(* PLC project MQTT, CODESYS CODESYS V3.5 SP14, author Stefan Dreyer *)
(* stored: creationDateTime 2019-02-05T05:32:10.3765761, version 1.0.0.0, modificationDateTime 2019-02-04T05:34:23.4609065, organization Stefan Dreyer *)
(* MQTT Stuff
Using some cool stuff of OSCAT libs.
see oscat.de

more to describe *)

{attribute 'qualified_only'}
{attribute 'strict'}
TYPE INSERT_SPLIT_RETURN : (INSERT_NOT_VALID := 0, INSERT_DONE, INSERT_PENDING, INSERT_ERROR);
END_TYPE

TYPE MESSAGETYPE : (CONNECT := 16#10, CONNACK := 16#20, PUBLISH := 16#30, PUBACK := 16#40, PUBREC := 16#50, PUBREL := 16#60, PUBCOMP := 16#70, SUBSCRIBE := 16#80, SUBACK := 16#90, UNSUBSCRIBE := 16#A0, UNSUBACK := 16#B0, PINGREQ := 16#C0, PINGRESP := 16#D0, DISCONNECT := 16#E0) BYTE;
END_TYPE

{attribute 'qualified_only'}
{attribute 'strict'}
TYPE PROG_NUM : (Publish, Subscribe, ParseIncomming, MoveBuffer, ParsePublish, GetBufferFreePos, GetSplitTopic, DESTROY_HANDLE_MQTT, DESTROY_SPLIT_TOPIC, STATE_MASHINE_IN, STATE_MASHINE_OUT, SendOutData, SendInData, SendOutDataInsertTopic, SendOutDataInsertPayload);
END_TYPE

{attribute 'qualified_only'}
{attribute 'strict'}
TYPE PUSHOVER_SOUND : (Standart := 1);
END_TYPE

TYPE QoS : (AtMostOnce := 2#0, AtLeastOnce := 2#1, ExactlyOnce := 2#10, Fail := 2#10000000) BYTE;
END_TYPE

{attribute 'qualified_only'}
{attribute 'strict'}
TYPE STEPS_IN : (WAIT_DATA := 0, SEND_PUBACK, SEND_PUBREC, WAIT_PUBREL, SEND_PUBCOMP);
END_TYPE

{attribute 'qualified_only'}
{attribute 'strict'}
TYPE STEPS_OUT : (WAIT_DATA := 0, SEND_PUBLSIH, WAIT_PUBREC, SEND_PUBREL, WAIT_PUBCOMP, WAIT_PUBACK, WAIT_PINGRESP, SEND_SUBSCRIBE, WAIT_SUBACK, SEND_UNSUBSCRIBE, WAIT_UNSUBACK);
END_TYPE

{attribute 'qualified_only'}
{attribute 'strict'}
TYPE TOPIC_MATCH : (TOPIC_MATCHES := 1, TOPIC_DONT_MATCHES := 2) BYTE;
END_TYPE

{attribute 'qualified_only'}
{attribute 'strict'}
TYPE TOPIC_VALID : (TOPIC_UNTESTED := 0, TOPIC_VALID := 2, TOPIC_NOT_VALID := 1, TOPIC_NO_TEST := 3) BYTE;
END_TYPE

(* this data is passed to a subscription callback *)
TYPE CALLBACK_DATA : STRUCT
  PayloadString : POINTER TO STRING;  (* the Payload String *)
  Payload : POINTER TO BYTE;  (* pointer to binary payload *)
  PayloadSize : UDINT;  (* size of binary payload *)
  TopicOut : POINTER TO STRING;  (* here you get the compleete recived topic string *)
  TopicOutSplit : POINTER TO SPLIT_TOPIC;  (* split topic.... *)
  PayloadIsString : BOOL;  (* Payload is string *)
END_STRUCT;
END_TYPE

{attribute 'enable_dynamic_creation'}
TYPE CALLBACK_INSTANCES : STRUCT
  callback : MQTT_SUBSCRIBE_CALLBACK;
  next : POINTER TO CALLBACK_INSTANCES;
  last : BOOL := TRUE;
END_STRUCT;
END_TYPE

TYPE LIST_ALLVALUES_CALLBACK_DATA : STRUCT
  VarTYPE : CommonTypesAndFunctions.VAR_TYPES;
  Target : CommonTypesAndFunctions.ALL_TYPES_UNION_POINTER;
  SubTopic : POINTER TO STRING;  (* pointer to last subtopic or Payload Data to compare with *)
END_STRUCT;
END_TYPE

TYPE LIST_STRING_CALLBACK_DATA : STRUCT
  Target : POINTER TO STRING;  (* pointer to target string *)
  SubTopic : POINTER TO STRING;  (* pointer to last subtopic or Payload Data to compare with *)
END_STRUCT;
END_TYPE

TYPE MQTT_SUBSCRIBE_CALLBACKS : STRUCT
  Callback : MQTT_SUBSCRIBE_CALLBACK;
  FbId : UINT;
  ExpectingString : BOOL;  (* expecting string *)
  SplitTopic : POINTER TO HandleSplitTopic;
  free : BOOL := TRUE;  (* set to false if slot is aquired by an subscription *)
END_STRUCT;
END_TYPE

(* here the maximum sizes of paylod and topics are defined if dynamic low init of split topic is used, don't care about MaxTopicElementSize *)
TYPE COM_CONFIG : STRUCT
  MaxPayloadSize : UDINT := 2000;  (* max payload size *)
  MaxTopicLevels : UINT := 25;  (* max topic levels *)
  MaxTopicElementSize : UINT := 255;  (* Max Topic elemt size *)
END_STRUCT;
END_TYPE

TYPE DATA_FROM_BROKER : STRUCT
  MqttTopic : POINTER TO STRING;  (* use array in size of network buffer to split message dynamic, maybe not ... best is dynamic mammory.... or use an array of Pointer.... or callbacks so lets try to buffer public messages and releas one per cycle to application... now we try dynamic memmory.... MQTT Topic from Broker *)
  Topics : POINTER TO SPLIT_TOPIC;
  MqttPayload : POINTER TO BYTE;  (* MQTT Payload for Broker Payload from broker --> Pointer *)
  MqttPayloadSize : UDINT;  (* Payload size *)
  MessageType : MESSAGETYPE;  (* MQTT Message Type *)
  DataRecived : BOOL;  (* Data recived *)
END_STRUCT;
END_TYPE

TYPE DATA_TO_BROKER : STRUCT
  PaketData : PAKET_DATA;  (* Data of Paket *)
END_STRUCT;
END_TYPE

(* contro struct between HANDLE_MQTT and MQTT_CONTROL *)
TYPE MQTT_COM : STRUCT
  S_BUF : NETWORK_BUFFER;
  R_BUF : NETWORK_BUFFER;
  MQTT_CON : BOOL;  (* if falling edge close with disconnect packet *)
  MQTT_ABORT : BOOL;  (* if using this to disconnect, don't send disconnect paket.... *)
  MQTT_URL : STRING(OSCAT_BASIC.STRING_LENGTH);
  MQTT_PACKET_NO : WORD;
  TIMEOUT : TIME;
  TLS : BOOL;  (* DNS_IP4 : DWORD; set to true if you want to use TLS *)
  TLS_CONFIG : POINTER TO CommonTypesAndFunctions.TLS_CONFIG := 0;  (* data to TLS stuff *)
  MQTT_RCV_STATE : BYTE;  (* 0= non 1= recived 2= error *)
  ERROR_C : DWORD;
  ERROR_T : BYTE;
  CLIENT_ID : STRING(23);  (* CONNECT_TO_LOCALHOST:BOOL; *)
  CLIENT_WILL_TOPIC : STRING(255);  (* Topic vof will message after client id *)
  CLIENT_WILL_MESSAGE_DEAD : STRING(255);
  CLIENT_WILL_RETAIN : BOOL := TRUE;
  BROKER_USER : STRING(254);
  BROKER_PASSWORD : STRING(254);
  MQTT_NO_AWNSER : BOOL;  (* pakte wihout request-- return to recivestate 1 *)
END_STRUCT;
END_TYPE

TYPE MQTT_IN_DATA : STRUCT
  step : STEPS_IN;
  PaketID : WORD;
  WaitsForBuffFree : ULINT;
  TimeOut : ton;
  TimeOutStarted : BOOL;
  PUBLISHOrder : UINT;
  PUBCOMPOrder : UINT;
  QoS : QoS;
  CountPubrecRepeat : UINT;
END_STRUCT;
END_TYPE

TYPE MQTT_IN_OUT : STRUCT
  handleFB : POINTER TO HANDLE_MQTT;  (* pointer to handle FB *)
  In : POINTER TO PAKET_DATA;
  InFree : BOOL := TRUE;  (* in free, true if free *)
  TDI : CommonTypesAndFunctions.TIME_DATE_IMPULS_DATA;  (* time, date, impulse... *)
  TLS_CONFIG : POINTER TO CommonTypesAndFunctions.TLS_CONFIG := 0;  (* TLS stuff data *)
  BROKER_CONNECTED : BOOL;
  FB_NO_AUTO : UINT;
  FB_NO_AUTO_COUNT : UINT;  (* FBs count *)
  FB_NO_AUTO_TOKEN : UINT := 1;  (* FB Token *)
  COM_CONFIG : COM_CONFIG;  (* config for boot up *)
  ClientID : STRING(23) := 'CODESYS_MQTT';  (* client ID, only chars 0123456789abcdefghijklmnopqrstuvwxyzABCDEFGHIJKLMNOPQRSTUVWXYZ" System never can be anonymos *)
  WillTopicBase : STRING(255) := 'MQTTWill';
  ClientWillTopic : STRING(30) := 'DEAD';
  ClientWillMessage : STRING(30) := 'DIED';
  dynMemUsage : UDINT;  (* usage of dynamic RAM *)
  disconnectOnBufferOverflow : BOOL;  (* set this to one if you want the client to act like the standardt says if set to one and we receve mor publish pakets than we can handle, QoS 0 packets are lost and QoS 1 and 2 packets have to be repeaded by he broker *)
END_STRUCT;
END_TYPE

TYPE MQTT_INFO : STRUCT
  MQTT_CONNECTED : BOOL;
  MQTT_ERROR : STRING(OSCAT_BASIC.STRING_LENGTH);
END_STRUCT;
END_TYPE

TYPE MQTT_OUT_DATA : STRUCT
  InDataFromFb : POINTER TO PAKET_DATA;
  step : STEPS_OUT;
  WaitsForBuffFree : ULINT;
  PUBRECOrder : UINT;
  TimeOut : ton;
  TimeOutStarted : BOOL;
  PUBLISHOrder : UINT;
  PUBRELRepeatCounter : UINT;
END_STRUCT;
END_TYPE

TYPE PAKET_DATA : STRUCT
  MqttTopic : POINTER TO STRING;  (* MQTT Topic for Broker *)
  MqttTopicLength : UINT;  (* Topic length *)
  MqttPayload : POINTER TO BYTE;  (* MQTT Payload for Broker *)
  MqttPayloadLength : UDINT;  (* Payload length *)
  MessageType : MESSAGETYPE;  (* MQTT Message Type *)
  MessageQoS : QoS;  (* MQTT QoS *)
  SubackQoS : QoS;  (* SUCACK QoS Response *)
  MessageRetain : BOOL;  (* MQTT reatin *)
  DUP : BOOL;  (* Retry of paket *)
  PaketId : WORD;  (* PakatID for header *)
  FbId : UINT;  (* ID of MQTT FB to store or of request to Broker *)
  SendSucsess : BOOL;  (* Send was succsessfull *)
  Callback : MQTT_SUBSCRIBE_CALLBACK;  (* Callback FB for subscription *)
  SplitTopic : POINTER TO HandleSplitTopic;  (* split topic for subscribe *)
  CallbackError : BOOL;  (* errore registering the callback *)
  ExpectingString : BOOL;  (* Expecting String *)
END_STRUCT;
END_TYPE

TYPE PUSHOVER_DATA : STRUCT
  Trigger : POINTER TO BOOL;
  Topic : POINTER TO STRING;
  Payload : POINTER TO STRING;
  Prio : USINT;
  Sound : PUSHOVER_SOUND;
  IsConfig : BOOL;
  R_T : R_TRIG;
  NeedToPush : BOOL;
  Negate : BOOL;
END_STRUCT;
END_TYPE

(* used for test cases... *)
TYPE RECIVE_PAKET : STRUCT
  MqttTopic : STRING(2000);  (* MQTT Topic *)
  MqttPayload : STRING(2000);  (* MQTT Payload *)
END_STRUCT;
END_TYPE

TYPE REMAINING_LENGTH_RETURN : STRUCT
  RemainingLength : UDINT;
  IndexAfterRemainingLength : UINT;
  Error : BOOL;
  BuffToSmall : BOOL;  (* not all bytes of remaining length in buffer... *)
  SizeRemainingLength : USINT;  (* size of remaining length *)
END_STRUCT;
END_TYPE

TYPE SEND_INFOS : STRUCT
  SubscribeIndex : UINT;  (* this index is to be subscribed *)
  SubscribeNeeded : BOOL := FALSE;
  SubscribeBlocking : BOOL;
  UnsubscribeIndex : UINT;  (* this index is to be subscribed *)
  UnsubscribeNeeded : BOOL := FALSE;
  UnsubscribeBlocking : BOOL;
  PublishBlocking : BOOL;  (* this index is to be published *)
  PublishBlockingIndex : UINT;
  PingIndex : UINT;  (* this index is to be published *)
  PingNeeded : BOOL;
END_STRUCT;
END_TYPE

TYPE SPLIT_TOPIC : STRUCT
  Topics : POINTER TO POINTER TO STRING;  (* this is going to be a pointer to a array of pointer to stings *)
  ValidFields : UINT;  (* count of vailid fields in the array *)
END_STRUCT;
END_TYPE

{attribute 'qualified_only'}
VAR_GLOBAL CONSTANT  (* MyConstants *)
  QoS_BUFFER_SIZE : UINT := 50;
  FB_BUFFER_SIZE : UINT := 5000;
  _COM_PAYLOAD_SIZE : UINT := 256;
  _MAX_TOPIC_LEVEL_SIZE : UINT := 255;  (* _COM_STRING_SIZE:UINT:=COM_PAYLOAD_SIZE; *)
  _MAX_PARTS_AT_TOPIC : INT := 25;
  _SQL_DATA_BUFFER_SIZE : UINT := 200;
  NETWORK_BUFFER_LONG_SIZE : UINT := 4095;
  KEEP_ALIVE_TIME : DWORD := 8;
  SENDING_TIMEOUT : TIME := TIME#4s0ms;
  REPEAT_TIMEOUT : TIME := TIME#2s0ms;
  REORDER_VALUE : UINT := 50000;  (* 50000 *)
  SUBSTRACTION_VALUE : UINT := 30000;  (* 20000 *)
  _COUNT_SUBTOPIC_FROM_BROKER : UINT := 25;
  MAX_PUBREL_REPEATS : UINT := 10;
END_VAR

{attribute 'qualified_only'}
VAR_GLOBAL  (* GVL_MQTT *)
  ProgNum : PROG_NUM;  (* Last Progamm stat for debug timeout exception *)
END_VAR

INTERFACE MQTT_SUBSCRIBE_CALLBACK
METHOD PublishRecived : BOOL
  VAR_INPUT
    Data : CALLBACK_DATA;  (* Collection of recived Data *)
  END_VAR
END_METHOD
END_INTERFACE

PROGRAM Doku

            (*

Hello There,

with this library you are able to send and recvice MQTT paket on all QoS levels 0-2.

Use Pubish to publish data(Strings and binary),

Use subscribe to recive MQTT data. On Subscribe you can tell the FB if you are expecting an String as data, so you will get one on the pointer output.

How to use you can see in the example and testCase FB. This is my Test Case an it does up to 100 send and recives per second on an raspberry PI 1+ connectet to an mosquitto broker on an 
windows 10 maschine.

If you find errors, or anny instability, tell me, i will have a look.

TLS works fine without certificates.

This Projekt i using some parts of the grat OSCAT libs, so take a look at oscat.de

Greatings 

*)
          
END_PROGRAM

FUNCTION_BLOCK TestOutOfTheBoxNoTLS
  VAR_INPUT
    client : STRING := 'test.mosquitto.org:1883';  (* test.mosquitto.org *)
  END_VAR
  VAR
    MQTTClient : HANDLE_MQTT;
    MQTT_IN_OUT : MQTT_IN_OUT;
    MQTTInfo : MQTT_INFO;
    publish : MQTTPublish;
    subscribe : MQTTSubscribe;
    ReciveSubscribeTopic : STRING(255);
    ReciveSubscribePayloadTick : STRING(255);
    ReciveSubscribePayloadState : STRING(255);
    State : MQTTState;
    init : BOOL;
    varSend : BOOL;
    timerSend : ton;
    t1 : ton;
    t2 : ton;
    Payload : STRING;
    StringCallback : ListStringCallback;  (* the method PublishReceved() is call when an publsih packet form the broker is recived. *)
    CallBackTargets : ARRAY[0..1] OF LIST_STRING_CALLBACK_DATA := [(Target := ADR(ReciveSubscribePayloadState), SubTopic := ADR('State')), (Target := ADR(ReciveSubscribePayloadTick), SubTopic := ADR('Tick'))];  (* the array contains the targets and sub topics for recive *)
  END_VAR

            //here init is done
IF NOT init THEN
	init := TRUE;
	MQTT_IN_OUT.ClientID := CONCAT('CodesysMqtt',TO_STRING(TICKS.GetTick(xDummy:= TRUE)));
	publish.SetMqttInOut(MQTT_IN_OUT:= ADR(MQTT_IN_OUT));
	subscribe.SetMqttInOut(MQTT_IN_OUT:= ADR(MQTT_IN_OUT));
	//init state FB, so you only have to call state();without parameters... 
	State.Init(
	State:= ADR(t1.Q), 
	Topic:= ADR('CODESYS-MQTT-BY-SD/State'), 
	StateName:= ADR(''), 
	StateValueOn:= ADR('On'), 
	StateValueOff:= ADR('Off'), 
	MQTT_IN_OUT:= ADR(MQTT_IN_OUT), 
	QoS:= QoS.ExactlyOnce, 
	RetainMqtt:= TRUE);
	StringCallback.InitAsSplitTopic(ListData := ADR(CallBackTargets), LengthOfData:= 2);

END_IF
//timer for repeating packets
timerSend(in := NOT varSend, PT := T#2S);
varSend := timerSend.Q; 
t1(IN:= NOT t2.Q, PT:= T#1S, );
t2(IN:= t1.Q, PT:= T#1S, );
//call of MQTT client
MQTTClient(
	MQTT_INFO:= MQTTInfo, 
	MQTT_IN_OUT:= MQTT_IN_OUT, 
	ENABLE:= TRUE, 
	URL:= client, 
	TIMEOUT:= T#5S, 
	TLS:= FALSE);
//build payload
IF varSend THEN
	Payload:= TO_STRING(TICKS.GetTick(xDummy:= TRUE));
END_IF
//Publish Payload
publish(
	Topic:= ADR('CODESYS-MQTT-BY-SD/Tick'), 
	PayloadString:= ADR(Payload), 
	PublishAsString:= TRUE, 
	QoSIn:= QoS.ExactlyOnce, 
	MRetain:= TRUE, 
	send:= varSend);
//Subscribe to topic
subscribe(
	Subscribe:= TRUE, 
	Topic:= ADR('CODESYS-MQTT-BY-SD/#'), 
	QoSSubscribe:= QoS.ExactlyOnce, 
	ExpectingString:= TRUE,
	Callback:= StringCallback);


//call of state FB
State();
          
END_FUNCTION_BLOCK

FUNCTION_BLOCK TestOutOfTheBoxTLS
  VAR_INPUT
    client : STRING := 'test.mosquitto.org:8883';  (* test.mosquitto.org *)
  END_VAR
  VAR
    MQTTClient : HANDLE_MQTT;
    MQTT_IN_OUT : MQTT_IN_OUT;
    MQTTInfo : MQTT_INFO;
    publish : MQTTPublish;
    subscribe : MQTTSubscribe;
    ReciveSubscribeTopic : STRING(255);
    ReciveSubscribePayloadTick : STRING(255);
    ReciveSubscribePayloadState : STRING(255);
    State : MQTTState;
    init : BOOL;
    varSend : BOOL;
    timerSend : ton;
    t1 : ton;
    t2 : ton;
    Payload : STRING;
    StringCallback : ListStringCallback;  (* the method PublishReceved() is call when an publsih packet form the broker is recived. *)
    CallBackTargets : ARRAY[0..1] OF LIST_STRING_CALLBACK_DATA := [(Target := ADR(ReciveSubscribePayloadState), SubTopic := ADR('State')), (Target := ADR(ReciveSubscribePayloadTick), SubTopic := ADR('Tick'))];  (* the array contains the targets and sub topics for recive *)
    TLS_CONFIG : CommonTypesAndFunctions.TLS_CONFIG;
  END_VAR

            //here init is done
IF NOT init THEN
	init := TRUE;
	MQTT_IN_OUT.ClientID := CONCAT('CodesysMqtt',TO_STRING(TICKS.GetTick(xDummy:= TRUE)));
	publish.SetMqttInOut(MQTT_IN_OUT:= ADR(MQTT_IN_OUT));
	subscribe.SetMqttInOut(MQTT_IN_OUT:= ADR(MQTT_IN_OUT));
	//init state FB, so you only have to call state();without parameters... 
	State.Init(
	State:= ADR(t1.Q), 
	Topic:= ADR('CODESYS-MQTT-BY-SD/State'), 
	StateName:= ADR(''), 
	StateValueOn:= ADR('On'), 
	StateValueOff:= ADR('Off'), 
	MQTT_IN_OUT:= ADR(MQTT_IN_OUT), 
	QoS:= QoS.ExactlyOnce, 
	RetainMqtt:= TRUE);
	StringCallback.InitAsSplitTopic(ListData := ADR(CallBackTargets), LengthOfData:= 2);
	MQTT_IN_OUT.TLS_CONFIG := ADR(TLS_CONFIG);
END_IF
//timer for repeating packets
timerSend(in := NOT varSend, PT := T#2S);
varSend := timerSend.Q; 
t1(IN:= NOT t2.Q, PT:= T#1S, );
t2(IN:= t1.Q, PT:= T#1S, );
//call of MQTT client
MQTTClient(
	MQTT_INFO:= MQTTInfo, 
	MQTT_IN_OUT:= MQTT_IN_OUT, 
	ENABLE:= TRUE, 
	URL:= client, 
	TIMEOUT:= T#5S, 
	TLS:= TRUE);
//build payload
IF varSend THEN
	Payload:= TO_STRING(TICKS.GetTick(xDummy:= TRUE));
END_IF
//Publish Payload
publish(
	Topic:= ADR('CODESYS-MQTT-BY-SD/Tick'), 
	PayloadString:= ADR(Payload), 
	PublishAsString:= TRUE, 
	QoSIn:= QoS.ExactlyOnce, 
	MRetain:= TRUE, 
	send:= varSend);
//Subscribe to topic	
subscribe(
	Subscribe:= TRUE, 
	Topic:= ADR('CODESYS-MQTT-BY-SD/#'), 
	QoSSubscribe:= QoS.ExactlyOnce, 
	ExpectingString:= TRUE,
	Callback:= StringCallback);


//call of state FB
State();
          
END_FUNCTION_BLOCK

(* true if levels the same *)
FUNCTION CheckTopicLevel : BOOL
  VAR_INPUT
    s1 : POINTER TO STRING;  (* String from Broker *)
    s2 : POINTER TO STRING;  (* Subscribe String *)
  END_VAR
  VAR
    LenS1 : UINT;
  END_VAR

            CheckTopicLevel := FALSE;
//test Wildcard
IF (s2^[0] = CommonTypesAndFunctions.GetChar(in:= '+')) THEN //(s2[0] = GetChar(in:= '#')) OR  don't check # here
	CheckTopicLevel := TRUE;
	RETURN;	
END_IF
LenS1 := CommonTypesAndFunctions.len(STR:= s1); 
IF (LenS1 <> CommonTypesAndFunctions.len(STR:= s2)) THEN 
	RETURN;
END_IF//if len not eval then return
IF (CommonTypesAndFunctions.find(STR1:= s1, STR2:= s2) >= 0) OR (LenS1 = 0)THEN
	CheckTopicLevel := TRUE;
END_IF
          
END_FUNCTION

FUNCTION DoRemainingLength : USINT
  VAR_INPUT
    buffer : POINTER TO BYTE;
    RemainingLength : UINT;
  END_VAR
  VAR
    LocalLength : LINT;
    LocalBuffer : ARRAY[0..3] OF BYTE;
    BufferIndex : UINT := 0;
    TmpByte : BYTE;
  END_VAR

            //check if we have to move data for inserting remaining length
//borders are given in the mqtt doku
//
IF RemainingLength <= 128 THEN
	buffer[1] := UINT_TO_BYTE(RemainingLength);
	DoRemainingLength := 0;
ELSE
	LocalLength := RemainingLength;
	REPEAT
		TmpByte := LINT_TO_BYTE(LocalLength MOD 128);
		LocalLength := LocalLength / 128;
		IF LocalLength > 0 THEN
			TmpByte := TmpByte OR 128;
		END_IF
		LocalBuffer[BufferIndex] := TmpByte; 
		BufferIndex := BufferIndex +1;
	UNTIL 
		LocalLength <= 0 
	END_REPEAT
	//now move mem	
	//buffer index points to NEXT field, so sub 1
	MEM.MemMove(pSource:= buffer+2, pDestination:= buffer + 2 + BufferIndex - 1 , uiNumberOfBytes:= RemainingLength);
	CASE BufferIndex OF
		2: 	buffer[1]:= LocalBuffer[0];
			buffer[2]:= LocalBuffer[1];
			DoRemainingLength := 1;
		3:	buffer[1]:= LocalBuffer[0];
			buffer[2]:= LocalBuffer[1];
			buffer[3]:= LocalBuffer[2];
			DoRemainingLength := 2;
		4:	buffer[1]:= LocalBuffer[0];
			buffer[2]:= LocalBuffer[1];
			buffer[3]:= LocalBuffer[2];
			buffer[4]:= LocalBuffer[3];
			DoRemainingLength := 3;
		
	END_CASE
	
END_IF

          
END_FUNCTION

(* here no move of data, call remainig length bevor moving topic and paylod, use this for borders are given in the mqtt doku use this for publish pakets *)
FUNCTION DoRemainingLengthBevor : USINT
  VAR_INPUT
    buffer : POINTER TO BYTE;  (* points to start of buffer, not to start of remainig length! *)
    SizeTopic : UDINT;
    SizePayload : UDINT;
    InQoS : QoS;
  END_VAR
  VAR
    RemainingLength : UDINT;
    LocalLength : LINT;
    LocalBuffer : ARRAY[0..3] OF BYTE;
    BufferIndex : UINT := 0;
    TmpByte : BYTE;
  END_VAR

            
	
RemainingLength := SizeTopic + SizePayload;
	
RemainingLength := RemainingLength + 2;//add topic size encoding space
IF NOT (InQoS = QoS.AtMostOnce) THEN
	RemainingLength := RemainingLength + 2;//add space for paket identifier
END_IF

IF RemainingLength <= 128 THEN
	buffer[1] := UDINT_TO_BYTE(RemainingLength);
	DoRemainingLengthBevor := 0;
ELSE
	LocalLength := RemainingLength;
	REPEAT
		TmpByte := LINT_TO_BYTE(LocalLength MOD 128);
		LocalLength := LocalLength / 128;
		IF LocalLength > 0 THEN
			TmpByte := TmpByte OR 128;
		END_IF
		LocalBuffer[BufferIndex] := TmpByte; 
		BufferIndex := BufferIndex +1;
	UNTIL 
		LocalLength <= 0 
	END_REPEAT
	CASE BufferIndex OF
		2: 	buffer[1]:= LocalBuffer[0];
			buffer[2]:= LocalBuffer[1];
			DoRemainingLengthBevor := 1;
		3:	buffer[1]:= LocalBuffer[0];
			buffer[2]:= LocalBuffer[1];
			buffer[3]:= LocalBuffer[2];
			DoRemainingLengthBevor := 2;
		4:	buffer[1]:= LocalBuffer[0];
			buffer[2]:= LocalBuffer[1];
			buffer[3]:= LocalBuffer[2];
			buffer[4]:= LocalBuffer[3];
			DoRemainingLengthBevor := 3;
		
	END_CASE
	
END_IF

          
END_FUNCTION

FUNCTION GetRemainingLength : REMAINING_LENGTH_RETURN
  VAR_INPUT
    Buff : POINTER TO BYTE;  (* Pointer to Buffer *)
    pos : UINT;  (* Start of data in Buffer *)
    BuffSize : UDINT;
  END_VAR
  VAR
    BufferIndex : UINT := 1;
    Multipler : UDINT := 1;
    TmpByte : BYTE;
  END_VAR

            GetRemainingLength.Error := FALSE;
GetRemainingLength.SizeRemainingLength:= 0;

GetRemainingLength.Error := FALSE;
BufferIndex := pos + 1;
REPEAT
	IF BufferIndex > (BuffSize - 1) THEN
		GetRemainingLength.BuffToSmall := TRUE;
	ELSE
		TmpByte := Buff[BufferIndex];
		BufferIndex := BufferIndex + 1;
		GetRemainingLength.RemainingLength := GetRemainingLength.RemainingLength + (TmpByte AND 127) * Multipler;
		Multipler := Multipler *128;
		IF Multipler > 128*128*128 THEN
			GetRemainingLength.RemainingLength := 0;//lengt 0 if broken
			GetRemainingLength.Error := TRUE;
		END_IF
	END_IF
	GetRemainingLength.SizeRemainingLength := GetRemainingLength.SizeRemainingLength + 1;
UNTIL
	(TmpByte AND 128) = 0 OR GetRemainingLength.RemainingLength = 0 OR GetRemainingLength.BuffToSmall
END_REPEAT
GetRemainingLength.IndexAfterRemainingLength := BufferIndex;
          
END_FUNCTION

FUNCTION InitMQTTValue : BOOL
  VAR_INPUT
    DataArray : POINTER TO CommonTypesAndFunctions.PWConfigs;
    CountOfArray : UINT;
    ValueToMQTTArray : POINTER TO MQTTValue;
    MQTT_IN_OUT : POINTER TO MQTT_IN_OUT;
  END_VAR
  VAR
    i : UINT;
  END_VAR

            FOR i := 0 TO CountOfArray - 1 DO
	IF DataArray[i].NeedsMQTT THEN
		ValueToMQTTArray[i].Init(
			Topic:= DataArray[i].MQTTTopic, 
			ValueName:= DataArray[i].MQTTName, 
			ValuePointer:= DataArray[i].PointerTo, 
			ValueType:= DataArray[i].ValueType, 
			ValueDiff:= DataArray[i].MQTTDiff, 
			MQTT_IN_OUT:= MQTT_IN_OUT, 
			DecimalPlace:= DataArray[i].MQTTDezimal, 
			QoS:= DataArray[i].MQTTQoS, 
			RetainMqtt:= DataArray[i].MQTTRetain, 
			MinTime:= DataArray[i].MQTTTime);
	END_IF
END_FOR
          
END_FUNCTION

(* returnds new pos in buff *)
FUNCTION InsertStringToBufferAndLength : UINT
  VAR_INPUT
    Str : POINTER TO STRING;
    buff : POINTER TO BYTE;  (* address to buffer *)
    pos : UINT;  (* Start to insert *)
  END_VAR
  VAR
    length : UINT;
  END_VAR

            length := CommonTypesAndFunctions.LEN(Str);
buff[pos]:= OSCAT_BASIC.BYTE_OF_DWORD(in:= length, N:= 1);
buff[pos+1]:= OSCAT_BASIC.BYTE_OF_DWORD(in:= length, N:= 0);

MEM.MemMove(pSource:= str, pDestination:= ADR(buff[pos+2]), uiNumberOfBytes:= length);
InsertStringToBufferAndLength := pos + length + 2;
          
END_FUNCTION

(* this FB collects instances of FB with the MQTT_SUBSCRIBE_CALLBACK interface. then you can pass a instance of this FB to a subscription FB to call all of your FBs to a specific subscription topic, in this call you can check if the packet was for your instance. If your instance methode call return true, the the FB exits the loop an so you may save cycle time. MEmory for instance references are created dynamic, so no restriction by library *)
FUNCTION_BLOCK CallbackCollector IMPLEMENTS MQTT_SUBSCRIBE_CALLBACK
  VAR
    first : CALLBACK_INSTANCES;
    firstHit : BOOL := TRUE;
  END_VAR

            
          

METHOD put : BOOL
  VAR_INPUT
    instance : MQTT_SUBSCRIBE_CALLBACK;
  END_VAR
  VAR
    aktElement : POINTER TO CALLBACK_INSTANCES;
  END_VAR
                  IF firstHit THEN
	firstHit := FALSE;
	first.callback := instance;
	RETURN;
END_IF
//first find last element
aktElement := ADR(first);

WHILE NOT aktElement^.last DO
	aktElement := aktElement^.next;
END_WHILE
{info 'semaphore'}
aktElement^.next := __NEW(CALLBACK_INSTANCES);
aktElement^.last := FALSE;
aktElement := aktElement^.next;
aktElement^.callback := instance;
aktElement^.last := TRUE;
                
END_METHOD

METHOD PublishRecived : BOOL
  VAR_INPUT
    Data : CALLBACK_DATA;  (* Collection of recived Data *)
  END_VAR
  VAR
    element : POINTER TO CALLBACK_INSTANCES;
    loop : BOOL := TRUE;
  END_VAR
                  IF firstHit THEN
	//no callback avalebal
	RETURN;
END_IF
element := ADR(first);


WHILE loop DO
	IF element^.callback.PublishRecived(Data := Data) THEN
		PublishRecived := TRUE;
		RETURN;
	END_IF
	IF element^.last THEN
		loop := FALSE;
	ELSE
		element := element^.next;
	END_IF
END_WHILE

                
END_METHOD

(* destroy all dynamic content *)
METHOD destroy : BOOL
  VAR
    aktElement : POINTER TO CALLBACK_INSTANCES;
    nextElement : POINTER TO CALLBACK_INSTANCES;
  END_VAR
                  IF firstHit THEN
	//no dyn memory used...
	RETURN;
END_IF
aktElement := ADR(first);

WHILE NOT nextElement^.last DO
	nextElement := aktElement^.next;
	__DELETE(aktElement);
	aktElement := nextElement; 
END_WHILE
__DELETE(aktElement);
                
END_METHOD

METHOD FB_Exit : BOOL
  VAR_INPUT
    bInCopyCode : BOOL;  (* TRUE: the exit method is called in order to leave the instance which will be copied afterwards (online change). *)
  END_VAR
                  destroy();
                
END_METHOD
END_FUNCTION_BLOCK

FUNCTION_BLOCK ReciveString IMPLEMENTS MQTT_SUBSCRIBE_CALLBACK
  VAR_OUTPUT
    MQTTRecived : STRING(255);  (* your desired payload... *)
  END_VAR
  VAR
    splitTopic : BOOL;  (* if set to true we search the instance name in the lowest topic *)
    splitPayload : BOOL;  (* if set to true we search the instance name in Payload separatet by the split char *)
    SplitPayloadChar : BYTE;  (* an this is the split char... *)
    MyCompString : POINTER TO STRING;  (* compare with this... *)
    MyReturnHit : BOOL;  (* if set to true and hit we will return true, else false... *)
  END_VAR

            
          

METHOD PublishRecived : BOOL
  VAR_INPUT
    Data : CALLBACK_DATA;  (* Collection of recived Data *)
  END_VAR
  VAR
    StrPt : POINTER TO STRING;
  END_VAR
                  // no we can check if the topic/payload fits to my instance name.... 

//now search the right topic 
IF splitTopic THEN
	
	IF CommonTypesAndFunctions.StrEquals(str1:= Data.TopicOutSplit^.Topics[Data.TopicOutSplit^.ValidFields - 1], str2:= MyCompString) THEN
		MQTTRecived := Data.PayloadString^;
		PublishRecived := MyReturnHit;
	END_IF

END_IF

//now look into the payload
IF splitPayload THEN
	
	IF CommonTypesAndFunctions.StrEqualsAtStartWithDelimiter(str1:= MyCompString, str2:= Data.PayloadString, delimiter:= SplitPayloadChar) THEN
		//now search split char
		StrPt := Data.PayloadString;
		StrPt := StrPt + TO_DWORD(CommonTypesAndFunctions.find(str1 := StrPt, str2:= ADR(SplitPayloadChar))) + 1;
		MQTTRecived := StrPt^;
		PublishRecived := MyReturnHit;
	END_IF
END_IF

                
END_METHOD

METHOD initAsFindTopic : BOOL
  VAR_INPUT
    compString : POINTER TO STRING;  (* this i'm searching *)
    returnHit : BOOL;  (* if set to true and hit we will return true, else false... *)
  END_VAR
                  
splitPayload := FALSE;
splitTopic := TRUE;
MyCompString := compString;
MyReturnHit := returnHit;
                
END_METHOD

METHOD initAsFindPayload : BOOL
  VAR_INPUT
    splitChar : STRING;  (* only first char is selected *)
    compString : POINTER TO STRING;  (* this i'm searching *)
    returnHit : BOOL;  (* if set to true and hit we will return true, else false... *)
  END_VAR
                  
splitPayload := TRUE;
splitTopic := FALSE;

SplitPayloadChar := CommonTypesAndFunctions.GetChar(in:= splitChar);
MyCompString := compString;
MyReturnHit := returnHit;
                
END_METHOD
END_FUNCTION_BLOCK

FUNCTION_BLOCK ReciveValue IMPLEMENTS MQTT_SUBSCRIBE_CALLBACK
  VAR_OUTPUT
    MQTTRecived : CommonTypesAndFunctions.ALL_TYPES_UNION;  (* your desired payload... *)
  END_VAR
  VAR
    TargetPointer : CommonTypesAndFunctions.ALL_TYPES_UNION_POINTER;  (* pointer to target *)
    MyValueTyp : CommonTypesAndFunctions.VAR_TYPES;  (* Target var type *)
    splitTopic : BOOL;  (* if set to true we search the instance name in the lowest topic *)
    splitPayload : BOOL;  (* if set to true we search the instance name in Payload separatet by the split char *)
    SplitPayloadChar : BYTE;  (* an this is the split char... *)
    MyCompString : POINTER TO STRING;  (* compare with this... *)
    MyReturnHit : BOOL;  (* if set to true and hit we will return true, else false... *)
  END_VAR

            
          

METHOD PublishRecived : BOOL
  VAR_INPUT
    Data : CALLBACK_DATA;  (* Collection of recived Data *)
  END_VAR
  VAR
    StrPt : POINTER TO STRING;
  END_VAR
                  IF splitTopic THEN
	//now search the right topic 
	IF CommonTypesAndFunctions.StrEquals(str1:= Data.TopicOutSplit^.Topics[Data.TopicOutSplit^.ValidFields - 1], str2:= MyCompString) THEN
		CommonTypesAndFunctions.GetValueFromStringPt(TypeOfValue:= MyValueTyp ,Target:= TargetPointer, str:= DATA.PayloadString^);
		PublishRecived := MyReturnHit;
	END_IF
	
END_IF
IF splitPayload THEN
	
	IF CommonTypesAndFunctions.StrEqualsAtStartWithDelimiter(str1:= MyCompString, str2:= Data.PayloadString, delimiter:= SplitPayloadChar) THEN
		//now search split char
		StrPt := Data.PayloadString;
		StrPt := StrPt + TO_DWORD(CommonTypesAndFunctions.find(str1 := StrPt, str2:= ADR(SplitPayloadChar))) + 1;
		CommonTypesAndFunctions.GetValueFromStringPt(TypeOfValue:= MyValueTyp ,Target:= TargetPointer, str:= StrPt^);
		PublishRecived := MyReturnHit;
	END_IF
	
END_IF
                
END_METHOD

METHOD initAsFindPayload : BOOL
  VAR_INPUT
    splitChar : STRING;  (* only first char is selected *)
    compString : POINTER TO STRING;  (* this i'm searching *)
    ValueTyp : CommonTypesAndFunctions.VAR_TYPES;  (* this typ is my recived string *)
    returnHit : BOOL;  (* if set to true and hit we will return true, else false... *)
  END_VAR
                  
splitPayload := TRUE;
splitTopic := FALSE;

SplitPayloadChar := CommonTypesAndFunctions.GetChar(in:= splitChar);
MyCompString := compString;
MyValueTyp := ValueTyp;
makePointer();
MyReturnHit := returnHit;
                
END_METHOD

METHOD initAsFindTopic : BOOL
  VAR_INPUT
    compString : POINTER TO STRING;  (* this i'm searching *)
    ValueTyp : CommonTypesAndFunctions.VAR_TYPES;  (* this typ is my recived string *)
    returnHit : BOOL;  (* if set to true and hit we will return true, else false... *)
  END_VAR
                  
splitPayload := FALSE;
splitTopic := TRUE;
MyCompString := compString;
MyValueTyp := ValueTyp;
makePointer();
MyReturnHit := returnHit;
                
END_METHOD

METHOD makePointer : BOOL
                  TargetPointer := CommonTypesAndFunctions.MakeAllTypesPointer(fromWho:= adr(MQTTRecived), myType:= MyValueTyp);
                
END_METHOD
END_FUNCTION_BLOCK

(* this FB expects all values as a string, binary recive is not suported... Payload content is only value, no description, no special characters... *)
FUNCTION_BLOCK ListAllValuesCallback IMPLEMENTS MQTT_SUBSCRIBE_CALLBACK
  VAR
    MyListData : POINTER TO LIST_ALLVALUES_CALLBACK_DATA;
    MyLengthOfData : ULINT;
    ListSplitTopic : BOOL;
    ListSplitPayload : BOOL;
    SplitCharPayload : BYTE;
  END_VAR

            
          

METHOD PublishRecived : BOOL
  VAR_INPUT
    Data : CALLBACK_DATA;  (* Collection of recived Data *)
  END_VAR
  VAR
    i : ULINT;
    StrPt : POINTER TO STRING;
  END_VAR
                  IF ListSplitTopic THEN
	//now search the right topic 
	FOR i := 0 TO MyLengthOfData - 1 DO
		IF CommonTypesAndFunctions.StrEquals(str1:= Data.TopicOutSplit^.Topics[Data.TopicOutSplit^.ValidFields - 1], str2:= MyListData[i].SubTopic) THEN
			CommonTypesAndFunctions.GetValueFromStringPt(TypeOfValue:= MyListData[i].VarTYPE ,Target:= MyListData[i].Target, str:= DATA.PayloadString^);
		END_IF
	END_FOR
END_IF
IF ListSplitPayload THEN
	FOR i := 0 TO MyLengthOfData - 1 DO
		IF CommonTypesAndFunctions.StrEqualsAtStartWithDelimiter(str1:= MyListData[i].SubTopic, str2:= Data.PayloadString, delimiter:= SplitCharPayload) THEN
			//now search split char
			StrPt := Data.PayloadString;
			StrPt := StrPt + TO_DWORD(CommonTypesAndFunctions.find(str1 := StrPt, str2:= ADR(SplitCharPayload))) + 1;
			
			CommonTypesAndFunctions.GetValueFromStringPt(TypeOfValue:= MyListData[i].VarTYPE ,Target:= MyListData[i].Target, str:= StrPt^);
		END_IF
	END_FOR
	
END_IF
                
END_METHOD

METHOD InitAsSplitTopic : BOOL
  VAR_INPUT
    Data : POINTER TO LIST_ALLVALUES_CALLBACK_DATA;
    LengthOfData : ULINT;  (* Count of List Data *)
  END_VAR
                  MyListData := Data;
MyLengthOfData := LengthOfData;
ListSplitTopic := TRUE;
ListSplitPayload := FALSE;
                
END_METHOD

(* inits FB, callback methoth then checks if the payload ist the same in the first characters as in the template make sure to recive a string payload! *)
METHOD InitAsSplitPayload : BOOL
  VAR_INPUT
    Data : POINTER TO LIST_ALLVALUES_CALLBACK_DATA;
    LengthOfData : ULINT;  (* Count of List Data *)
    SplitChar : BYTE;  (* spliting character *)
  END_VAR
                  MyListData :=Data;
MyLengthOfData := LengthOfData;
ListSplitTopic := FALSE;
ListSplitPayload := TRUE;
SplitCharPayload := SplitChar;
                
END_METHOD
END_FUNCTION_BLOCK

FUNCTION_BLOCK ListStringCallback IMPLEMENTS MQTT_SUBSCRIBE_CALLBACK
  VAR
    MyListData : POINTER TO LIST_STRING_CALLBACK_DATA;
    MyLengthOfData : ULINT;
    ListSplitTopic : BOOL;
    ListSplitPayload : BOOL;
    SplitCharPayload : BYTE;
  END_VAR

            
          

METHOD PublishRecived : BOOL
  VAR_INPUT
    Data : CALLBACK_DATA;  (* Collection of recived Data *)
  END_VAR
  VAR
    i : ULINT;
    StrPt : POINTER TO STRING;
  END_VAR
                  //now search the right topic 
IF ListSplitTopic THEN
	FOR i := 0 TO MyLengthOfData - 1 DO
		IF CommonTypesAndFunctions.StrEquals(str1:= Data.TopicOutSplit^.Topics[Data.TopicOutSplit^.ValidFields - 1], str2:= MyListData[i].SubTopic) THEN
			MyListData[i].Target^ := Data.PayloadString^;
		END_IF
	END_FOR
END_IF

IF ListSplitPayload THEN
	FOR i := 0 TO MyLengthOfData - 1 DO
		IF CommonTypesAndFunctions.StrEqualsAtStartWithDelimiter(str1:= MyListData[i].SubTopic, str2:= Data.PayloadString, delimiter:= SplitCharPayload) THEN
			//now search split char
			StrPt := Data.PayloadString;
			StrPt := StrPt + TO_DWORD(CommonTypesAndFunctions.find(str1 := StrPt, str2:= ADR(SplitCharPayload))) + 1;
			MyListData[i].Target^ := StrPt^;
		END_IF
	END_FOR
	
END_IF

                
END_METHOD

(* ints FB to split packets at lowest payload level *)
METHOD InitAsSplitTopic : BOOL
  VAR_INPUT
    ListData : POINTER TO LIST_STRING_CALLBACK_DATA;
    LengthOfData : ULINT;  (* Count of List Data *)
  END_VAR
                  MyListData :=ListData;
MyLengthOfData := LengthOfData;
ListSplitTopic := TRUE;
ListSplitPayload := FALSE;

                
END_METHOD

(* inits FB, callback methoth then checks if the payload ist the same in the first characters as in the template make sure to recive a string payload! *)
METHOD InitAsSplitPayload : BOOL
  VAR_INPUT
    ListData : POINTER TO LIST_STRING_CALLBACK_DATA;
    LengthOfData : ULINT;  (* Count of List Data *)
    SplitChar : BYTE;  (* spliting character *)
  END_VAR
                  MyListData :=ListData;
MyLengthOfData := LengthOfData;
ListSplitTopic := FALSE;
ListSplitPayload := TRUE;
SplitCharPayload := SplitChar;
                
END_METHOD
END_FUNCTION_BLOCK

(* this FB expects all values as a string, binary recive is not suported... Payload content is only value, no description, no special characters... *)
FUNCTION_BLOCK AllValuesCallback IMPLEMENTS MQTT_SUBSCRIBE_CALLBACK
  VAR
    VarType : CommonTypesAndFunctions.VAR_TYPES;
    MyTarget : CommonTypesAndFunctions.ALL_TYPES_UNION_POINTER;
  END_VAR

            
          

METHOD PublishRecived : BOOL
  VAR_INPUT
    Data : CALLBACK_DATA;  (* Collection of recived Data *)
  END_VAR
                  CommonTypesAndFunctions.GetValueFromStringPt(TypeOfValue:= VarType,Target:= MyTarget, str:= DATA.PayloadString^);
                
END_METHOD

METHOD Init : BOOL
  VAR_INPUT
    SetType : CommonTypesAndFunctions.VAR_TYPES;
    Target : CommonTypesAndFunctions.ALL_TYPES_UNION_POINTER;
  END_VAR
                  VarType := SetType;
MyTarget := Target;

                
END_METHOD
END_FUNCTION_BLOCK

FUNCTION_BLOCK SingelStringCallback IMPLEMENTS MQTT_SUBSCRIBE_CALLBACK
  VAR
    MyPayload : POINTER TO STRING;
    MyTopic : POINTER TO STRING;
  END_VAR

            
          

METHOD PublishRecived : BOOL
  VAR_INPUT
    Data : CALLBACK_DATA;  (* Collection of recived Data *)
  END_VAR
                  MyPayload^ := Data.PayloadString^;
MyTopic^ := Data.TopicOut^;


                
END_METHOD

METHOD Init : BOOL
  VAR_INPUT
    payload : POINTER TO STRING;
    topic : POINTER TO STRING;
  END_VAR
                  MyTopic := topic;
MyPayload := payload;
                
END_METHOD
END_FUNCTION_BLOCK

FUNCTION_BLOCK ClientWrapper
  VAR_INPUT
    broker : STRING(255);
    connect : BOOL;
    tls : BOOL := FALSE;
    ClientID : STRING(255);
  END_VAR
  VAR_OUTPUT
    MQTT_IN_OUT : MQTT_IN_OUT;
    MQTTInfo : MQTT_INFO;
  END_VAR
  VAR
    MQTTClient : HANDLE_MQTT;
  END_VAR

            MQTT_IN_OUT.ClientID := ClientID;

MQTTClient(
	MQTT_INFO:= MQTTInfo, 
	MQTT_IN_OUT:= MQTT_IN_OUT, 
	ENABLE:= connect, 
	URL:= broker, 
	TIMEOUT:= T#5S, 
	TLS:= tls);
	
          
END_FUNCTION_BLOCK

(* var/log/mosquitto/mosquitto.log Messsages are not beeing repeatet, if timout for an answer then connection is canceled, new established and the publisher have to start new Start the command line subscriber: mosquitto_sub -v -t 'test/topic' mosquitto_sub -v -h test.mosquitto.org -t 'test/topic' sudo apt-get install tshark tshark -i 1 -a duration:60 -w /tmp/wlan.pcap debug / logging : mosquitto_sub -v -t '$SYS/#' sudo nano /etc/mosquitto/mosquitto.conf --> 'log_type all' Publish test message with the command line publisher: mosquitto_pub -t 'test/topic' -m 'helloWorld' change check free to InFbNo kopieren sudo cp /var/log/mosquitto/mosquitto.log /tmp/ zugriff sudo chmod -v a=r /tmp/mosquitto.log TODO: Take care of clean session, is enabled, do it paramable? layout publish recive buffer: recive publish buffer layout: 0 byte 3 of topic length of udint 1 byte 2 of topic length of udint 2 byte 1 of topic length of udint 3 byte 0 of topic length of udint 4+n Topic string without termination n byte 3 of payload length of udint n+1 byte 2 of payload length of udint n+2 byte 1 of payload length of udint n+3 byte 0 of payload length of udint n+4+x Payload *)
FUNCTION_BLOCK HANDLE_MQTT
  VAR_IN_OUT
    MQTT_INFO : MQTT_INFO;
    MQTT_IN_OUT : MQTT_IN_OUT;
  END_VAR
  VAR_INPUT
    ENABLE : BOOL;
    URL : STRING(OSCAT_BASIC.STRING_LENGTH);
    TIMEOUT : TIME;
    TLS : BOOL;
  END_VAR
  VAR_OUTPUT
    ERROR_C : DWORD;
    ERROR_T : BYTE;
  END_VAR
  VAR
    DT_MQTT : CommonTypesAndFunctions.TIME_DATE_IMPULS;
    MQTT_CONTROL : MQTT_CONTROL;
    step : INT;
    i1 : UINT;
    PingSlot : UINT;
    COM : MQTT_COM;
    TmpString : STRING(255);
    TimeoutConnection : TON;
    MqttsDoneIo : ULINT;
    CycleTime : DWORD;
    LastCycleTime : DWORD;
    NextPingTime : CAA.TICK;
    PingTime : CAA.TICK := ((MyConstants.KEEP_ALIVE_TIME * 1000) - 6000);  (* next ping after 6 seconds *)
    PingRequestet : BOOL;  (* Ping was sendet *)
    PingData : DATA_TO_BROKER;
    myFbNo : UINT;
    PubrelOrderIndexCounter : UINT;
    PubcompOrderIndexCounter : UINT;
    LogFile : CAA.HANDLE;  (* log file *)
    open : FILE.Open;
    write : FILE.Write;
    LogString : STRING(255);
    DebugFile : BOOL := FALSE;
    OutData : ARRAY[0..MyConstants.QoS_BUFFER_SIZE] OF MQTT_OUT_DATA;
    InData : ARRAY[0..MyConstants.QoS_BUFFER_SIZE] OF MQTT_IN_DATA;
    PublishSendListCount : UINT;
    PublishSendList : ARRAY[0..MyConstants.QoS_BUFFER_SIZE] OF UINT;
    PubrelSendListCount : UINT;
    PubrelSendList : ARRAY[0..MyConstants.QoS_BUFFER_SIZE] OF UINT;
    PubackSendListCount : UINT;
    PubackSendList : ARRAY[0..MyConstants.QoS_BUFFER_SIZE] OF UINT;
    PubrecSendListCount : UINT;
    PubrecSendList : ARRAY[0..MyConstants.QoS_BUFFER_SIZE] OF UINT;
    PubcompSendListCount : UINT;
    PubcompSendList : ARRAY[0..MyConstants.QoS_BUFFER_SIZE] OF UINT;
    RepeatedPublish : ULINT;  (* Repeted Publishs *)
    RepeatedPublishsAfterPubrel : ULINT;  (* Repeatet publishs afert ot much repeat of pubrel *)
    RepeatedPubrel : ULINT;  (* Repeted pubrel *)
    CountRepeatedPing : ULINT;  (* Repeted Ping *)
    CountRepeatedPingDisconnect : UINT;  (* Repeated pings untill disconnect *)
    PublishsUnacknowledged : UINT;  (* count of Publishs unacknowledged *)
    LastToBigTopic : STRING(255);  (* last part of 255 chars of to big paket topic *)
    CountToBigTopics : ULINT;  (* count of to big topics *)
    CountLengthErrors : ULINT;  (* Cont of ength Error Pakets *)
    CountRepeatPublishRecive : ULINT;  (* Count of repeatet publishs *)
    CountRecivedPublishs : ULINT;  (* Count Recived Publishs *)
    CountSendedPublishs : ULINT;  (* count sended publishs *)
    CountRepeatSubscribe : ULINT;  (* Count of repeated subscribs *)
    CountRepeatUnsubscribe : ULINT;  (* Count of repeated unsubscribs *)
    CountRepeatetPubrec : ULINT;  (* Count of repeatet pubrec *)
    CountOutputPublishCalled : ULINT;  (* Count of OutputPublish calls *)
    PUBREC_ERROR_ID_BUFFER : ARRAY[0..(PUBREC_ERROR_ID_BUFFER_SIZE - 1)] OF UINT;
    PUBREC_ERROR_INDEX : UINT;
    OutgoingPublishOrderIndexCounter : UINT;  (* send Publish order Index *)
    IncomingPublishOrderIndexCounter : UINT;  (* recive Publish order Index *)
    CountRecivePubrelUnknown : ULINT;  (* Recived Pubrel, Paket not found *)
    CountReciveUnsubackUnknown : ULINT;  (* Recived Unsuback, Paket not found *)
    CountReciveSubackUnknown : ULINT;  (* Recived Suback, Paket not found *)
    CountRecivePubackUnknown : ULINT;  (* Recived Puback, Paket not found *)
    CountRecivePubrecUnknown : ULINT;  (* Recived Pubrec, Paket not found *)
    CountRecivePubcompUnknown : ULINT;  (* Recived Pubcomp, Paket not found *)
    SendInfos : SEND_INFOS;
    CountOutSendNotFree : ULINT;
    CountInSendNotFree : ULINT;
    CountCantSendPublishBufferToFull : ULINT;
    CounterPublishSendForMonitor : UINT;
    PublishsSendPerSeconde : UINT;
    CounterPublishRecivedForMonitor : UINT;
    PublishsRecivedPerSeconde : UINT;
    NotKnownPaket : MESSAGETYPE;
    CountUnkownPaket : ULINT;
    LastPaktetForUnkownPaket : MESSAGETYPE;
    HelperLastPaktetForUnkownPaket : MESSAGETYPE;
    CountBufferMoves : ULINT;
    CountNothingSend : ULINT;
    CountConnectAttempt : ULINT;
    CountSplitTopicSizeExceeded : ULINT;  (* count of topic size exceeded *)
    CountWaitForRestOfPaket : ULINT;  (* PublishReciveBuffer:ARRAY[0..RECIVE_PUBLISH_BUFFER_SIZE]OF BYTE; PublishReciveBufferCount:UINT; PublishReciveBufferCountMax:UINT; PublishReciveTopicLengt:UDINT; PublishRecivePayloadLengt:UDINT; size of assignment in recive publish buffer PublishReciveBufferAssignment: UDINT; PublishReciveBufferAssignmentMax: UDINT; PublishReciveBufferCountFull:ULINT; *)
    CountResetBufferIn : ULINT;
    InBufferMoved : UINT;
    SendFree : BOOL;
    MySplitTopic : HandleSplitTopic;
    InsertSplitTopic : InsertSplitTopic;  (* PublishSplitetd: BOOL; *)
    InsertSplitPayload : InsertSplitPayload;
    StepBuildPublish : INT;
    StepBuildSubscribe : INT;
    StepBuildUnsubscribe : INT;
    SplitPublishBuffer : POINTER TO BYTE;  (* use this buffer for recived publish packets whos size exceded network buffer Size *)
    SplitPublishBufferSize : UDINT;
    SplitPublishLength : UDINT;
    MaxPublishPacketSize : UDINT;  (* output from buffer Don't write new data! SplitPublishLock:BOOL; *)
    PayloadMemorySize : DWORD;
    SubscribeCallbacks : ARRAY[0..(CALLBACKS_BUFFER_SIZE - 1)] OF MQTT_SUBSCRIBE_CALLBACKS;
    TopicMemorySize : DWORD;
    COM_CONFIG : COM_CONFIG;
    PublishSplited : BOOL;  (* BufferTopic:ARRAY[0..SIZEOF(COM.S_BUF.BUFFER)]OF BYTE;//doesn't need to be biger than network buffer, because is only used if full paket resits in network buffer BufferPayload:ARRAY[0..SIZEOF(COM.S_BUF.BUFFER)]OF BYTE; publish paket broken, waiting for more data *)
    DoDisconnect : BOOL;
    SendetBytes : ULINT;
    RecivedBytes : ULINT;
    InSlotsWorking : UINT;
    OutSlotsWorking : UINT;
    DynMemUsagePointer : POINTER TO UDINT;
    CallbacksFull : BOOL;  (* callbacks array full *)
  END_VAR
  VAR CONSTANT
    CALLBACKS_BUFFER_SIZE : UINT := 200;
    RECIVE_PUBLISH_BUFFER_SIZE : UINT := (NETWORK_BUFFER_LONG_SIZE * 2);
    TRANSMIT_BUFFER_SIZE : UINT := NETWORK_BUFFER_LONG_SIZE;
    SIZE_PUBREL : UINT := 4;
    SIZE_UNSUBACK : UINT := 4;
    SIZE_PINGRESP : UINT := 2;
    SIZE_PINGREQ : UINT := 2;
    SIZE_SUBACK : UINT := 5;
    SIZE_PUBACK : UINT := 4;
    SIZE_PUBREC : UINT := 4;
    SIZE_PUBCOMP : UINT := 4;
    SIZE_PAKET_BUFFER_HEADER : UINT := 4;
    PUBREC_ERROR_ID_BUFFER_SIZE : UINT := 100;
    MAX_PING_REPEATS : UINT := 10;
    SPLIT_PUBLISH_BUFFER_ADDITIONAL_RAM : UINT := 17;
    COUNT_MAX_PUBREC_REPEAT_TO_DISCHARGE : UINT := 20;
  END_VAR

            //first organisize FB nums and FB Tokens...
myFbNo := MQTT_IN_OUT.FB_NO_AUTO + 1;
MQTT_IN_OUT.FB_NO_AUTO_COUNT := myFbNo;
//reset token
IF MQTT_IN_OUT.FB_NO_AUTO_TOKEN >= myFbNo - 1 THEN
	MQTT_IN_OUT.FB_NO_AUTO_TOKEN := 1;
END_IF
IF MQTT_INFO.MQTT_CONNECTED THEN
	SendFree := COM.S_BUF.SIZE = 0;	
END_IF

MQTT_IN_OUT.FB_NO_AUTO := 0;//reset FB number
CycleTime := OSCAT_BASIC.T_PLC_MS() - LastCycleTime;
LastCycleTime := OSCAT_BASIC.T_PLC_MS();
//get system time and so one
DT_MQTT(
	TDI_Data:= MQTT_IN_OUT.TDI);
	
TimeoutConnection(IN:= step = 10, PT:= T#5S);

IF DebugFile THEN
		//open log file
		open(
	xExecute:= TRUE, 
	sFileName:= '/tmp/mqtt.log', 
	eFileMode:= 0, 
	xExclusive:= TRUE, 
	hFile=> LogFile);
END_IF

CASE step OF

	00:	IF ENABLE THEN
			MQTT_IN_OUT.handleFB := THIS;
			PublishsUnacknowledged := 0;
			PUBREC_ERROR_INDEX := 0;
			CountRepeatedPingDisconnect := 0;
			SendetBytes := 0;
			RecivedBytes := 0;		
			PublishSplited := FALSE;
			DoDisconnect := FALSE;
			SendInfos.PingNeeded := FALSE;
			SendInfos.SubscribeNeeded := FALSE;
			SendInfos.UnsubscribeNeeded := FALSE;
			StepBuildPublish := 0;
			StepBuildSubscribe := 0;
			StepBuildUnsubscribe := 0;
			InsertSplitTopic.reset();
			InsertSplitPayload.reset();
			CountConnectAttempt := CountConnectAttempt + 1;
			DynMemUsagePointer := ADR(MQTT_IN_OUT.dynMemUsage);
			COM.MQTT_URL := URL;
			COM.TIMEOUT := TIMEOUT;
			COM.CLIENT_ID := MQTT_IN_OUT.ClientID;
			COM.TLS := TLS;
			COM.TLS_CONFIG := MQTT_IN_OUT.TLS_CONFIG;
			ResetPingTime();
			//build will topic
			{info 'check build will topic'}
			TmpString := MQTT_IN_OUT.WillTopicBase;
			TmpString := Standard.CONCAT(STR1:= TmpString, '/');
			TmpString := Standard.CONCAT(STR1:= TmpString, STR2:= COM.CLIENT_ID);
			TmpString := Standard.CONCAT(STR1:= TmpString, '/');
			TmpString := Standard.CONCAT(STR1:= TmpString, MQTT_IN_OUT.ClientWillTopic);
			COM.CLIENT_WILL_TOPIC := TmpString;
			COM.CLIENT_WILL_MESSAGE_DEAD := MQTT_IN_OUT.ClientWillMessage;
			COM_CONFIG := MQTT_IN_OUT.COM_CONFIG;
			FOR i1 := 0 TO MyConstants.QoS_BUFFER_SIZE - 1 DO
				//reset in slots
				InData[i1].step := STEPS_IN.WAIT_DATA;
				OutData[i1].step := STEPS_OUT.WAIT_DATA;
			END_FOR
			//reset callbacks
			FOR i1 := 0 TO CALLBACKS_BUFFER_SIZE - 1 DO
				SubscribeCallbacks[i1].free := TRUE; 
			END_FOR
			MySplitTopic.FullInit(TopicsLevelInit:= COM_CONFIG.MaxTopicLevels, SplitElementSizeInit:= COM_CONFIG.MaxTopicElementSize, dynMemUsageInit:= ADR(MQTT_IN_OUT.dynMemUsage));
			//MQTT_IN_OUT.OUT.Topics := SplitTopic.GetSplitTopic(); 
			PayloadMemorySize := COM_CONFIG.MaxPayloadSize;
			{warning disable C0033}
			TopicMemorySize := COM_CONFIG.MaxTopicElementSize * COM_CONFIG.MaxTopicLevels;
			MaxPublishPacketSize := (COM_CONFIG.MaxTopicElementSize * COM_CONFIG.MaxTopicLevels) + PayloadMemorySize;
			{info 'semaphore'}
			//SplitPublishBuffer  := SysMem23.SysMemAlloc(dwSize:= MaxPublishPacketSize + SPLIT_PUBLISH_BUFFER_ADDITIONAL_RAM);//some additional bytes for paket overhead and termination
			SplitPublishBuffer  := __NEW(BYTE, (MaxPublishPacketSize + SPLIT_PUBLISH_BUFFER_ADDITIONAL_RAM));//some additional bytes for paket overhead and termination
			MQTT_IN_OUT.dynMemUsage := MQTT_IN_OUT.dynMemUsage + MaxPublishPacketSize + SPLIT_PUBLISH_BUFFER_ADDITIONAL_RAM;
			{warning restore C0033}

			step := 10;
			COM.MQTT_CON := TRUE;
				
					
		
		END_IF;
	10:	IF MQTT_INFO.MQTT_CONNECTED THEN
			step := 40;
		END_IF;
		IF TimeoutConnection.Q THEN
			step := 0;//reset steps
			destroy();
		END_IF
	40:	
		IF PublishSplited THEN
			MergeSplitedPublish(MQTT_IN_OUT:= ADR(MQTT_IN_OUT));
		END_IF	
		ParseIncoming(MQTT_IN_OUT:= ADR(MQTT_IN_OUT));
		PublishSendListCount := 0;
		PubrelSendListCount := 0;
		PubackSendListCount := 0;
		PubrecSendListCount := 0;
		PubcompSendListCount := 0;
		StateMashineIn(MQTT_IN_OUT:= ADR(MQTT_IN_OUT));
		StateMashineOut( MQTT_IN_OUT:= ADR(MQTT_IN_OUT));
		
		SendOutData(MQTT_IN_OUT:= ADR(MQTT_IN_OUT));
		SendInData(MQTT_IN_OUT:= ADR(MQTT_IN_OUT));
	
		IF MQTT_IN_OUT.TDI.IMP THEN
			PublishsSendPerSeconde := CounterPublishSendForMonitor;
			CounterPublishSendForMonitor := 0;
			PublishsRecivedPerSeconde := CounterPublishRecivedForMonitor;
			CounterPublishRecivedForMonitor := 0;
		END_IF
		IF COM.S_BUF.SIZE = 0 THEN
			CountNothingSend := CountNothingSend + 1;
		END_IF
		IF NOT ENABLE THEN 	(* beenden? *)
			step := 50;
			
		END_IF;
		IF DoDisconnect THEN
			DoDisconnect := FALSE;
			//here hard disconnect
			COM.MQTT_CON := FALSE; (* MQTT Verbindung beenden *)
			COM.MQTT_ABORT := TRUE;
			
			step := 60;
		END_IF

(* ~~~~~~~~~~~~~~~~~~~~~~ *)

50: 
	COM.MQTT_CON := FALSE; (* MQTT Verbindung beenden *)
	
	step := 60;//wait for disconnect
60:
	IF MQTT_INFO.MQTT_CONNECTED = FALSE THEN
		destroy();
		step := 0;
		
	END_IF
END_CASE;



(* ########################## *)

IF CountRepeatedPingDisconnect > MAX_PING_REPEATS THEN
	DoDisconnect := TRUE;
END_IF


SendetBytes := SendetBytes + COM.S_BUF.SIZE;
MQTT_CONTROL(COM:= COM, INFO:=MQTT_INFO);
RecivedBytes := RecivedBytes + COM.R_BUF.SIZE;
ERROR_C := COM.ERROR_C;
ERROR_T := COM.ERROR_T;
//handl ping telegram
IF NextPingTime < TICKS.GetTick(xDummy:= TRUE) AND NOT PingRequestet AND ENABLE THEN
	
	MakePingPaket(MQTT_IN_OUT := MQTT_IN_OUT);
	
END_IF

IF COM.ERROR_T > BYTE#0 THEN  (* FEHLER *)
	step := 0;
END_IF;
//put status to local clients
MQTT_IN_OUT.BROKER_CONNECTED := MQTT_INFO.MQTT_CONNECTED;
(* ########################## *)

(* revision history


*)
          

METHOD ResetPingTime
                  NextPingTime := PingTime + TICKS.GetTick(xDummy:= TRUE);
CountRepeatedPingDisconnect := 0;
                
END_METHOD

METHOD MakePingPaket
  VAR_IN_OUT
    MQTT_IN_OUT : MQTT_IN_OUT;
  END_VAR
                  IF MQTT_IN_OUT.InFree THEN 
	MQTT_IN_OUT.IN := ADR(PingData); //set request
	PingData.PaketData.MessageType := MESSAGETYPE.PINGREQ;
	PingData.PaketData.FbId := myFbNo;
	MQTT_IN_OUT.InFree := FALSE;
	PingRequestet := TRUE;
END_IF

                
END_METHOD

METHOD StateMashineOut
  VAR_INPUT
    MQTT_IN_OUT : POINTER TO MQTT_IN_OUT;  (* StepData:POINTER TO MQTT_OUT_DATA; *)
  END_VAR
  VAR
    i : UINT;
    j : UINT;
    tmpLowest : UINT;
    minIndex : UINT;
    UnsubscribeLastHighest : UINT := 16#FFFF;
    SubscribeLastHighest : UINT := 16#FFFF;
    RecivePaketID : WORD;  (* PublishLastHighest : UINT := 16#FFFF; PubrelLastHighest : UINT := 16#FFFF; *)
    RecivePakteType : BYTE;
    TempSlotsWorking : UINT;
  END_VAR
                  (*need a token for coordinate send of pakets....
prio for Awnser and repeat pakets bevor new publish
dont use token, just send paket with next publish index*)
//get paket id
RecivePaketID := DWORD_TO_WORD(OSCAT_BASIC.DWORD_OF_BYTE(B3:= 0, B2:= 0, B1:= COM.R_BUF.BUFFER[2], B0:= COM.R_BUF.BUFFER[3]));
RecivePakteType := COM.R_BUF.BUFFER[0] AND 16#F0; 

GVL_MQTT.ProgNum := PROG_NUM.STATE_MASHINE_OUT;
PublishSendListCount := 0;
PubrelSendListCount := 0;

TempSlotsWorking := 0;
FOR i := 0 TO MyConstants.QoS_BUFFER_SIZE - 1 DO
	//do Timers...
	OutData[i].TimeOut(IN:= OutData[i].TimeOutStarted, PT:= MyConstants.REPEAT_TIMEOUT);
	CASE OutData[i].step OF
		
		STEPS_OUT.WAIT_DATA:
			OutData[i].TimeOutStarted := FALSE;
		IF NOT MQTT_IN_OUT^.InFree THEN//new Data from FBs
			MQTT_IN_OUT^.InFree := TRUE;
			OutData[i].InDataFromFb := MQTT_IN_OUT^.In;//set Data
			//Pakte id = slot + 1....
			OutData[i].InDataFromFb^.PaketId := i + 1;
			CASE OutData[i].InDataFromFb^.MessageType OF
				MESSAGETYPE.PUBLISH:
					OutgoingPublishOrderIndexCounter := OutgoingPublishOrderIndexCounter + 1;
					OutData[i].PUBLISHOrder :=  OutgoingPublishOrderIndexCounter;
					OutData[i].step := STEPS_OUT.SEND_PUBLSIH;
					CountSendedPublishs := CountSendedPublishs + 1;
					CounterPublishSendForMonitor := CounterPublishSendForMonitor + 1;
					OutData[i].PUBRELRepeatCounter := 0;
				MESSAGETYPE.PINGREQ:
					OutData[i].step := STEPS_OUT.WAIT_PINGRESP;
					SendInfos.PingNeeded := TRUE;
					SendInfos.PingIndex := i;
					PingSlot := i;
				//we only sending one subscription per subscribe paket....
				MESSAGETYPE.SUBSCRIBE:
					//check if we have a slot free for subscription
					FOR j := 0 TO CALLBACKS_BUFFER_SIZE - 1 DO
						IF SubscribeCallbacks[j].free THEN
							OutData[i].step := STEPS_OUT.SEND_SUBSCRIBE;
							CallbacksFull := FALSE;
							EXIT;
						END_IF
					END_FOR
					IF j = CALLBACKS_BUFFER_SIZE THEN
						//no free slot
						MQTT_IN_OUT^.In^.CallbackError := TRUE;
						CallbacksFull := TRUE;
					END_IF
				MESSAGETYPE.UNSUBSCRIBE:
					OutData[i].step := STEPS_OUT.SEND_UNSUBSCRIBE;
			END_CASE
			
		END_IF
		
		STEPS_OUT.WAIT_PINGRESP:
			IF OutData[i].TimeOutStarted AND OutData[i].TimeOut.Q AND NOT SendInfos.PingNeeded THEN
				//timeout, need repead
				SendInfos.PingNeeded := TRUE;
				SendInfos.PingIndex := i;
				CountRepeatedPing := CountRepeatedPing + 1; 
				CountRepeatedPingDisconnect := CountRepeatedPingDisconnect + 1;
				OutData[i].TimeOutStarted := FALSE;
			END_IF
		STEPS_OUT.SEND_UNSUBSCRIBE:
			//check if my paket ID is the lowest to send it
			IF OutData[i].InDataFromFb^.PaketId < UnsubscribeLastHighest AND NOT SendInfos.UnsubscribeNeeded THEN
				SendInfos.UnsubscribeIndex := i;
				SendInfos.UnsubscribeNeeded := TRUE;
				UnsubscribeLastHighest := OutData[i].InDataFromFb^.PaketId;
			END_IF	
		STEPS_OUT.WAIT_UNSUBACK:
			IF OutData[i].TimeOutStarted AND OutData[i].TimeOut.Q THEN
				//timeout, need repead
				OutData[i].step := STEPS_OUT.SEND_UNSUBSCRIBE;//repeat subscribe
				CountRepeatUnsubscribe := CountRepeatUnsubscribe + 1;
				OutData[i].TimeOutStarted := FALSE;
			END_IF
		STEPS_OUT.SEND_SUBSCRIBE:
			//check if my paket ID is the lowest to send it
			IF OutData[i].InDataFromFb^.PaketId < SubscribeLastHighest AND NOT SendInfos.SubscribeNeeded THEN
				SendInfos.SubscribeIndex := i;
				SendInfos.SubscribeNeeded := TRUE;
				SubscribeLastHighest := OutData[i].InDataFromFb^.PaketId;
			END_IF	
		STEPS_OUT.WAIT_SUBACK:
			IF OutData[i].TimeOutStarted AND OutData[i].TimeOut.Q THEN
				//timeout, need repead
				OutData[i].step := STEPS_OUT.SEND_SUBSCRIBE;//repeat subscribe
				CountRepeatSubscribe := CountRepeatSubscribe + 1;
				OutData[i].TimeOutStarted := FALSE;
			END_IF
			
		STEPS_OUT.SEND_PUBLSIH:
			PublishSendList[PublishSendListCount] := i;
			PublishSendListCount := PublishSendListCount + 1;
			
		STEPS_OUT.WAIT_PUBACK:
			IF OutData[i].TimeOutStarted AND OutData[i].TimeOut.Q THEN
				//timeout, need repead
				OutData[i].InDataFromFb^.DUP := TRUE;
				OutData[i].step := STEPS_OUT.SEND_PUBLSIH;//repeat publish
				RepeatedPublish := RepeatedPublish + 1;
				OutData[i].TimeOutStarted := FALSE;
			END_IF
			
		STEPS_OUT.WAIT_PUBREC:
			IF OutData[i].TimeOutStarted AND OutData[i].TimeOut.Q THEN
				//timeout, need repead
				OutData[i].InDataFromFb^.DUP := TRUE;
				OutData[i].step := STEPS_OUT.SEND_PUBLSIH;//repeat publish
				RepeatedPublish := RepeatedPublish + 1;
				OutData[i].TimeOutStarted := FALSE;
			END_IF
			
		STEPS_OUT.SEND_PUBREL:
			PubrelSendList[PubrelSendListCount] := i;
			PubrelSendListCount := PubrelSendListCount + 1;
			
		STEPS_OUT.WAIT_PUBCOMP:
			IF OutData[i].TimeOutStarted AND OutData[i].TimeOut.Q THEN
				//timeout, need repead
				OutData[i].step := STEPS_OUT.SEND_PUBREL;//repeat pubrel
				RepeatedPubrel := RepeatedPubrel + 1;
				OutData[i].TimeOutStarted := FALSE;
				OutData[i].PUBRELRepeatCounter := OutData[i].PUBRELRepeatCounter + 1;
				IF OutData[i].PUBRELRepeatCounter >= MyConstants.MAX_PUBREL_REPEATS THEN
					OutData[i].PUBRELRepeatCounter := 0;
					//resend publish
					OutData[i].step := STEPS_OUT.SEND_PUBLSIH;
					OutData[i].InDataFromFb^.DUP := TRUE;
					RepeatedPublishsAfterPubrel := RepeatedPublishsAfterPubrel + 1;
				END_IF
			END_IF
		IF NOT (OutData[i].step = STEPS_OUT.WAIT_DATA) THEN
			TempSlotsWorking := TempSlotsWorking + 1;
		END_IF
	END_CASE
	//make sure timer is set to 0 if timeout resetet
	OutData[i].TimeOut(IN:= OutData[i].TimeOutStarted, PT:= MyConstants.REPEAT_TIMEOUT);
END_FOR

//now sort the arrays...
IF PublishSendListCount > 1 THEN
	FOR i := 0 TO PublishSendListCount - 1 DO
		tmpLowest := 16#FFFF;
		minIndex := i;
		FOR j := i TO PublishSendListCount - 1 DO
			IF OutData[PublishSendList[j]].PUBLISHOrder < tmpLowest THEN
				minIndex := j;
				tmpLowest := OutData[PublishSendList[j]].PUBLISHOrder;
			END_IF
		END_FOR
		IF minIndex <> i THEN
			//hier tauschen
			j := PublishSendList[minIndex];
			PublishSendList[minIndex] := PublishSendList[i];
			PublishSendList[i] := j;
		END_IF
	END_FOR
END_IF

IF PubrelSendListCount > 1 THEN
	FOR i := 0 TO PubrelSendListCount - 1 DO
		tmpLowest := 16#FFFF;
		minIndex := i;
		FOR j := i TO PubrelSendListCount - 1 DO
			IF OutData[PubrelSendList[j]].PUBRECOrder < tmpLowest THEN
				minIndex := j;
				tmpLowest := OutData[PubrelSendList[j]].PUBRECOrder;
			END_IF
		END_FOR
		IF minIndex <> i THEN
			//hier tauschen
			j := PubrelSendList[minIndex];
			PubrelSendList[minIndex] := PubrelSendList[i];
			PubrelSendList[i] := j;
		END_IF
	END_FOR
END_IF

//Hamdel PubrelOrderIndexCounter
IF PubrelOrderIndexCounter > MyConstants.REORDER_VALUE THEN 
	//do it brute force, just sub 20000 to every value...
	FOR i := 0 TO MyConstants.QoS_BUFFER_SIZE - 1 DO
		OutData[i].PUBRECOrder := OutData[i].PUBRECOrder - MyConstants.SUBSTRACTION_VALUE;
	END_FOR
	PubrelOrderIndexCounter := MyConstants.REORDER_VALUE - MyConstants.SUBSTRACTION_VALUE + 1;
END_IF
//Hamdel PublishOrderIndexCounter
IF OutgoingPublishOrderIndexCounter > MyConstants.REORDER_VALUE THEN 
	//do it brute force, just sub 20000 to every value...
	FOR i := 0 TO MyConstants.QoS_BUFFER_SIZE - 1 DO
		OutData[i].PUBLISHOrder := OutData[i].PUBLISHOrder - MyConstants.SUBSTRACTION_VALUE;
	END_FOR
	OutgoingPublishOrderIndexCounter := MyConstants.REORDER_VALUE - MyConstants.SUBSTRACTION_VALUE + 1;
END_IF

OutSlotsWorking := TempSlotsWorking;
                
END_METHOD

METHOD StateMashineIn
  VAR_INPUT
    MQTT_IN_OUT : POINTER TO MQTT_IN_OUT;
  END_VAR
  VAR
    i : UINT;
    j : UINT;
    TempSlotsWorking : UINT;
    tmpLowest : UINT;
    minIndex : UINT;
  END_VAR
                  //RecivePakteType := COM.R_BUF.BUFFER[0] AND 16#F0;
GVL_MQTT.ProgNum := PROG_NUM.STATE_MASHINE_IN;
//Handle State Mashines
PubackSendListCount := 0;
PubrecSendListCount := 0;
PubcompSendListCount := 0;
TempSlotsWorking := 0;
FOR i := 0 TO MyConstants.QoS_BUFFER_SIZE - 1 DO
	//do Timers...
	InData[i].TimeOut(IN:= InData[i].TimeOutStarted, PT:= MyConstants.REPEAT_TIMEOUT);
	IF NOT (InData[i].step = STEPS_IN.WAIT_DATA) THEN
		TempSlotsWorking := TempSlotsWorking + 1;
	END_IF  
	CASE InData[i].step OF
		STEPS_IN.WAIT_DATA:;
		STEPS_IN.WAIT_PUBREL:
		IF InData[i].TimeOut.Q THEN
			InData[i].step := STEPS_IN.SEND_PUBREC;
			InData[i].TimeOutStarted := FALSE;
			CountRepeatetPubrec := CountRepeatetPubrec + 1;
			PUBREC_ERROR_ID_BUFFER[PUBREC_ERROR_INDEX] := InData[i].PaketID; 
			PUBREC_ERROR_INDEX := PUBREC_ERROR_INDEX + 1;
			InData[i].CountPubrecRepeat := InData[i].CountPubrecRepeat + 1;
			IF InData[i].CountPubrecRepeat > COUNT_MAX_PUBREC_REPEAT_TO_DISCHARGE THEN
				InData[i].CountPubrecRepeat := 0;
				InData[i].step := STEPS_IN.WAIT_DATA;
			END_IF
			IF PUBREC_ERROR_INDEX >= PUBREC_ERROR_ID_BUFFER_SIZE THEN
				PUBREC_ERROR_INDEX := 0;
			END_IF
		END_IF
		STEPS_IN.SEND_PUBACK:
			PubackSendList[PubackSendListCount] := i;
			PubackSendListCount := PubackSendListCount + 1;
			
		STEPS_IN.SEND_PUBREC:
			PubrecSendList[PubrecSendListCount] := i;
			PubrecSendListCount := PubrecSendListCount + 1;
		
		STEPS_IN.SEND_PUBCOMP:
			PubcompSendList[PubcompSendListCount] := i;
			PubcompSendListCount := PubcompSendListCount + 1;
		
	END_CASE
	//make sure timer is set to 0 if timeout resetet
	InData[i].TimeOut(IN:= InData[i].TimeOutStarted, PT:= MyConstants.REPEAT_TIMEOUT);
END_FOR


//now sort the arrays...
IF PubackSendListCount > 1 THEN
	FOR i := 0 TO PubackSendListCount - 1 DO
		tmpLowest := 16#FFFF;
		minIndex := i;
		FOR j := i TO PubackSendListCount - 1 DO
			IF InData[PubackSendList[j]].PUBLISHOrder < tmpLowest THEN
				minIndex := j;
				tmpLowest := InData[PubackSendList[j]].PUBLISHOrder;
			END_IF
		END_FOR
		IF minIndex <> i THEN
			//hier tauschen
			j := PubackSendList[minIndex];
			PubackSendList[minIndex] := PubackSendList[i];
			PubackSendList[i] := j;
		END_IF
	END_FOR
END_IF

IF PubrecSendListCount > 1 THEN
	FOR i := 0 TO PubrecSendListCount - 1 DO
		tmpLowest := 16#FFFF;
		minIndex := i;
		FOR j := i TO PubrecSendListCount - 1 DO
			IF InData[PubrecSendList[j]].PUBLISHOrder < tmpLowest THEN
				minIndex := j;
				tmpLowest := InData[PubrecSendList[j]].PUBLISHOrder;
			END_IF
		END_FOR
		IF minIndex <> i THEN
			//hier tauschen
			j := PubrecSendList[minIndex];
			PubrecSendList[minIndex] := PubrecSendList[i];
			PubrecSendList[i] := j;
		END_IF
	END_FOR
END_IF


IF PubcompSendListCount > 1 THEN
	FOR i := 0 TO PubcompSendListCount - 1 DO
		tmpLowest := 16#FFFF;
		minIndex := i;
		FOR j := i TO PubcompSendListCount - 1 DO
			IF InData[PubcompSendList[j]].PUBCOMPOrder < tmpLowest THEN
				minIndex := j;
				tmpLowest := InData[PubcompSendList[j]].PUBCOMPOrder;
			END_IF
		END_FOR
		IF minIndex <> i THEN
			//hier tauschen
			j := PubcompSendList[minIndex];
			PubcompSendList[minIndex] := PubcompSendList[i];
			PubcompSendList[i] := j;
		END_IF
	END_FOR
END_IF
//Hamdel PublishOrderIndexCounter
IF IncomingPublishOrderIndexCounter > MyConstants.REORDER_VALUE THEN 
	//do it brute force, just sub 20000 to every value...
	FOR i := 0 TO MyConstants.QoS_BUFFER_SIZE - 1 DO
		InData[i].PUBLISHOrder := InData[i].PUBLISHOrder - MyConstants.SUBSTRACTION_VALUE;
	END_FOR
	IncomingPublishOrderIndexCounter := MyConstants.REORDER_VALUE - MyConstants.SUBSTRACTION_VALUE + 1;
END_IF

//Hamdel PublishOrderIndexCounter
IF PubcompOrderIndexCounter > MyConstants.REORDER_VALUE THEN 
	//do it brute force, just sub 20000 to every value...
	FOR i := 0 TO MyConstants.QoS_BUFFER_SIZE - 1 DO
		InData[i].PUBCOMPOrder := InData[i].PUBCOMPOrder - MyConstants.SUBSTRACTION_VALUE;
	END_FOR
	PubcompOrderIndexCounter := MyConstants.REORDER_VALUE - MyConstants.SUBSTRACTION_VALUE + 1;
END_IF

InSlotsWorking := TempSlotsWorking;
                
END_METHOD

METHOD BuildPublishPaket : BOOL
  VAR_INPUT
    PaketData : POINTER TO PAKET_DATA;
  END_VAR
  VAR
    idx : UINT;
  END_VAR
                  (*now change to realy big topics and payloads, do that to big topics and payloads transmitted splitted*)

BuildPublishPaket := FALSE;
IF StepBuildPublish = 0 THEN
	StepBuildPublish := 10; 
END_IF

idx := COM.S_BUF.SIZE;
//check if buffer is big enought for control, remainig length, topic size....
IF StepBuildPublish = 10 THEN

	IF (6 + COM.S_BUF.SIZE)
		 > TRANSMIT_BUFFER_SIZE THEN//only check if header fits into buffer...
		 CountCantSendPublishBufferToFull := CountCantSendPublishBufferToFull + 1;
		RETURN;	
	END_IF
	COM.S_BUF.BUFFER[idx] := MESSAGETYPE.PUBLISH;//set type
	IF PaketData^.DUP THEN//insert DUP bit
		COM.S_BUF.BUFFER[idx] := COM.S_BUF.BUFFER[idx] OR 2#1000;
	END_IF 
	COM.S_BUF.BUFFER[idx] := COM.S_BUF.BUFFER[idx] OR SHL(PaketData^.MessageQoS,1);
	IF PaketData^.MessageRetain THEN
		COM.S_BUF.BUFFER[idx] := COM.S_BUF.BUFFER[idx] OR 2#1;
	END_IF
	//do remainig lenght... 

	idx := idx + 2 + DoRemainingLengthBevor(buffer:= ADR(COM.S_BUF.BUFFER[idx]), SizeTopic:= PaketData^.MqttTopicLength, SizePayload:= PaketData^.MqttPayloadLength, InQoS:= PaketData^.MessageQoS);

	StepBuildPublish := 20;
END_IF

IF StepBuildPublish = 20 THEN
	GVL_MQTT.ProgNum := PROG_NUM.SendOutDataInsertTopic;
	//insert topic
	InsertSplitTopic(
		topic:= PaketData^.MqttTopic, 
		len:= PaketData^.MqttTopicLength, 
		buff:= ADR(COM.S_BUF.BUFFER), 
		pos:= idx, 
		size:= NETWORK_BUFFER_LONG_SIZE);
	CASE InsertSplitTopic.state OF
		INSERT_SPLIT_RETURN.INSERT_DONE:
			StepBuildPublish := 30;
		INSERT_SPLIT_RETURN.INSERT_ERROR:
			StepBuildPublish := 0;
			InsertSplitTopic.reset();
			RETURN;
		INSERT_SPLIT_RETURN.INSERT_PENDING:
			//here do nothing, just wait
		ELSE
			InsertSplitTopic.reset();
			StepBuildPublish := 0;
			RETURN;
	END_CASE
	idx := InsertSplitTopic.new_pos;
END_IF
IF StepBuildPublish = 30 THEN
	IF PaketData^.MessageQoS > 0 THEN//QoS is more then 0
		IF (2 + idx)//insert paket identifier
		 < TRANSMIT_BUFFER_SIZE THEN//enough space for identifier?
			COM.S_BUF.BUFFER[idx] := OSCAT_BASIC.BYTE_OF_DWORD(in:= PaketData^.PaketId, N:= 1);
			idx := idx + 1;
			COM.S_BUF.BUFFER[idx] := OSCAT_BASIC.BYTE_OF_DWORD(in:= PaketData^.PaketId, N:= 0);
			idx := idx + 1;
			StepBuildPublish := 40;
		END_IF
	ELSE
		StepBuildPublish := 40;
	END_IF
END_IF

IF StepBuildPublish = 40 THEN
	GVL_MQTT.ProgNum := PROG_NUM.SendOutDataInsertPayload;
	//now insert payload
	IF PaketData^.MqttPayloadLength > 0 THEN
		//insert payload
		InsertSplitPayload(
			payload:= PaketData^.MqttPayload, 
			len:= PaketData^.MqttPayloadLength, 
			buff:= ADR(COM.S_BUF.BUFFER), 
			pos:= idx, 
			size:= NETWORK_BUFFER_LONG_SIZE);
		CASE InsertSplitPayload.state OF
			INSERT_SPLIT_RETURN.INSERT_DONE:
				StepBuildPublish := 0;
				BuildPublishPaket := TRUE;
			INSERT_SPLIT_RETURN.INSERT_ERROR:
				StepBuildPublish := 0;
				InsertSplitPayload.reset();
				RETURN;
			INSERT_SPLIT_RETURN.INSERT_PENDING:
				//here do nothing, just wait
				//or handle timeout....
			ELSE
				InsertSplitPayload.reset();
				StepBuildPublish := 0;
				RETURN;
		END_CASE
		idx := InsertSplitPayload.new_pos;
	ELSE
		StepBuildPublish := 0;
		BuildPublishPaket := TRUE;
	END_IF
END_IF
COM.S_BUF.SIZE := idx;

                
END_METHOD

METHOD MoveBufferForSplitPaket
  VAR_INPUT
    idx : UINT;
  END_VAR
  VAR
    BytesToMove : UINT;
  END_VAR
                  GVL_MQTT.ProgNum := PROG_NUM.MoveBuffer;
BytesToMove := COM.R_BUF.SIZE - idx;
CountBufferMoves := CountBufferMoves + 1;
MEM.MemMove(pSource:= ADR(com.R_BUF.BUFFER[idx]), pDestination:= ADR(com.R_BUF.BUFFER), uiNumberOfBytes:= BytesToMove);
COM.R_BUF.SIZE := BytesToMove;//manipulate size....

                
END_METHOD

METHOD BuildSubscribePaket : BOOL
  VAR_INPUT
    PaketData : POINTER TO PAKET_DATA;
  END_VAR
  VAR
    idx : UINT;
  END_VAR
                  BuildSubscribePaket := FALSE;
IF  StepBuildSubscribe = 0 THEN
	StepBuildSubscribe := 10;
END_IF

idx := COM.S_BUF.SIZE;
IF StepBuildSubscribe = 10 THEN
	IF (6 + COM.S_BUF.SIZE)
	 > TRANSMIT_BUFFER_SIZE THEN//only check if header fits into buffer...
		 RETURN;
	END_IF
	idx := COM.S_BUF.SIZE;
	COM.S_BUF.BUFFER[idx] := MESSAGETYPE.SUBSCRIBE OR 2#10;//set type, for 2#10 see subscribe doku
	idx := idx + 2 + DoRemainingLengthBevor(buffer:= ADR(COM.S_BUF.BUFFER[idx]), SizeTopic:= PaketData^.MqttTopicLength, SizePayload:= 1, InQoS:= QoS.AtLeastOnce);
	COM.S_BUF.BUFFER[idx] := OSCAT_BASIC.BYTE_OF_DWORD(in:= PaketData^.PaketId, N:= 1);
	idx := idx + 1;
	COM.S_BUF.BUFFER[idx] := OSCAT_BASIC.BYTE_OF_DWORD(in:= PaketData^.PaketId, N:= 0);
	idx := idx + 1;
	StepBuildSubscribe := 20;
END_IF


IF StepBuildSubscribe = 20 THEN
	//insert topic
	InsertSplitTopic(
		topic:= PaketData^.MqttTopic, 
		len:= PaketData^.MqttTopicLength, 
		buff:= ADR(COM.S_BUF.BUFFER), 
		pos:= idx, 
		size:= NETWORK_BUFFER_LONG_SIZE);
	CASE InsertSplitTopic.state OF
		INSERT_SPLIT_RETURN.INSERT_DONE:
			StepBuildSubscribe := 30;
		INSERT_SPLIT_RETURN.INSERT_ERROR:
			StepBuildSubscribe := 0;
			InsertSplitTopic.reset();
			RETURN;
		INSERT_SPLIT_RETURN.INSERT_PENDING:
			//here do nothing, just wait
		ELSE
			InsertSplitTopic.reset();
			StepBuildSubscribe := 0;
			RETURN;
	END_CASE
	idx := InsertSplitTopic.new_pos;
END_IF

IF StepBuildSubscribe = 30 THEN

	IF (1 + idx)
	 > TRANSMIT_BUFFER_SIZE THEN//only check if qos fits into buffer...
		 RETURN;
	 END_IF
	//insert QoS
	COM.S_BUF.BUFFER[idx] := PaketData^.MessageQoS;
	idx := idx + 1;
	StepBuildSubscribe := 0;
	BuildSubscribePaket := TRUE;
END_IF

COM.S_BUF.SIZE := idx;
                
END_METHOD

METHOD BuildUnsubscribePaket : BOOL
  VAR_INPUT
    PaketData : POINTER TO PAKET_DATA;
  END_VAR
  VAR
    idx : UINT;
  END_VAR
                  BuildUnsubscribePaket := FALSE;

IF  StepBuildUnsubscribe = 0 THEN
	StepBuildUnsubscribe := 10;
END_IF

idx := COM.S_BUF.SIZE;
IF StepBuildUnsubscribe = 10 THEN
	IF (6 + COM.S_BUF.SIZE)
	 > TRANSMIT_BUFFER_SIZE THEN//only check if header fits into buffer...
		 RETURN;
	END_IF
	idx := COM.S_BUF.SIZE;
	COM.S_BUF.BUFFER[idx] := MESSAGETYPE.UNSUBSCRIBE OR 2#10;//set type, for 2#10 see subscribe doku
	idx := idx + 2 + DoRemainingLengthBevor(buffer:= ADR(COM.S_BUF.BUFFER[idx]), SizeTopic:= PaketData^.MqttTopicLength, SizePayload:= 0, InQoS:= QoS.AtLeastOnce);
	COM.S_BUF.BUFFER[idx] := OSCAT_BASIC.BYTE_OF_DWORD(in:= PaketData^.PaketId, N:= 1);
	idx := idx + 1;
	COM.S_BUF.BUFFER[idx] := OSCAT_BASIC.BYTE_OF_DWORD(in:= PaketData^.PaketId, N:= 0);
	idx := idx + 1;
	StepBuildUnsubscribe := 20;
END_IF


IF StepBuildUnsubscribe = 20 THEN
	//insert topic
	InsertSplitTopic(
		topic:= PaketData^.MqttTopic, 
		len:= PaketData^.MqttTopicLength, 
		buff:= ADR(COM.S_BUF.BUFFER), 
		pos:= idx, 
		size:= NETWORK_BUFFER_LONG_SIZE);
	CASE InsertSplitTopic.state OF
		INSERT_SPLIT_RETURN.INSERT_DONE:
			StepBuildUnsubscribe := 0;
			BuildUnsubscribePaket := TRUE;
		INSERT_SPLIT_RETURN.INSERT_ERROR:
			StepBuildUnsubscribe := 0;
			InsertSplitTopic.reset();
			RETURN;
		INSERT_SPLIT_RETURN.INSERT_PENDING:
			//here do nothing, just wait
		ELSE
			InsertSplitTopic.reset();
			StepBuildUnsubscribe := 0;
			RETURN;
	END_CASE
	idx := InsertSplitTopic.new_pos;
END_IF

COM.S_BUF.SIZE := idx;

                
END_METHOD

METHOD SendOutData
  VAR_INPUT
    MQTT_IN_OUT : POINTER TO MQTT_IN_OUT;  (* StepData:POINTER TO MQTT_OUT_DATA; *)
  END_VAR
  VAR
    SomethingIsBlocking : BOOL;
    i : UINT;
  END_VAR
                  IF NOT SendFree THEN RETURN; END_IF
GVL_MQTT.ProgNum := PROG_NUM.SendOutData;

SomethingIsBlocking := SendInfos.PublishBlocking OR SendInfos.SubscribeBlocking OR SendInfos.UnsubscribeBlocking;

//Prio for Timeout Paket
IF  NOT (COM.S_BUF.SIZE + SIZE_PINGREQ > TRANSMIT_BUFFER_SIZE) AND SendInfos.PingNeeded AND NOT SomethingIsBlocking THEN
	SendInfos.PingNeeded := FALSE;
	COM.S_BUF.BUFFER[COM.S_BUF.SIZE] := MESSAGETYPE.PINGREQ;
	COM.S_BUF.BUFFER[COM.S_BUF.SIZE + 1] := 0;//no more length 	
	COM.S_BUF.SIZE := COM.S_BUF.SIZE + SIZE_PINGREQ;//small ping paket
	OutData[SendInfos.PingIndex].TimeOutStarted := TRUE;//start Timeout
END_IF
IF NOT COM.S_BUF.SIZE = 0 THEN 
	CountOutSendNotFree := CountOutSendNotFree + 1;
END_IF
//next Prio send Pubrel 
IF PubrelSendListCount > 0 AND NOT SomethingIsBlocking THEN
	FOR i := 0 TO PubrelSendListCount - 1 DO
		IF NOT (COM.S_BUF.SIZE + SIZE_PUBREL > TRANSMIT_BUFFER_SIZE) THEN
			//SendInfos.PubrelNeeded := FALSE;
			COM.S_BUF.BUFFER[COM.S_BUF.SIZE] := MESSAGETYPE.PUBREL OR 2#10;//set type and Reserved bits
			COM.S_BUF.BUFFER[COM.S_BUF.SIZE + 1] := 2;
			COM.S_BUF.BUFFER[COM.S_BUF.SIZE + 2] := OSCAT_BASIC.BYTE_OF_DWORD(in:= OutData[PubrelSendList[i]].InDataFromFb^.PaketId, N:= 1);
			COM.S_BUF.BUFFER[COM.S_BUF.SIZE + 3] := OSCAT_BASIC.BYTE_OF_DWORD(in:= OutData[PubrelSendList[i]].InDataFromFb^.PaketId, N:= 0);
			COM.S_BUF.SIZE := COM.S_BUF.SIZE + SIZE_PUBREL;
			OutData[PubrelSendList[i]].step := STEPS_OUT.WAIT_PUBCOMP;
			OutData[PubrelSendList[i]].TimeOutStarted := TRUE;//start Timeout			
		ELSE
			EXIT;
		END_IF 
	END_FOR
END_IF

//send Unsubscribe
IF SendInfos.UnsubscribeNeeded AND (NOT SomethingIsBlocking OR SendInfos.UnsubscribeBlocking) THEN
	IF NOT BuildUnsubscribePaket(PaketData:= OutData[SendInfos.UnsubscribeIndex].InDataFromFb) THEN
		SendInfos.UnsubscribeBlocking := TRUE;
	ELSE
		SendInfos.UnsubscribeBlocking := FALSE;
		SendInfos.UnsubscribeNeeded := FALSE;
		OutData[SendInfos.UnsubscribeIndex].TimeOutStarted := TRUE;
		OutData[SendInfos.UnsubscribeIndex].step := STEPS_OUT.WAIT_UNSUBACK;
	END_IF
END_IF

//send Subscribe
IF SendInfos.SubscribeNeeded AND (NOT SomethingIsBlocking OR SendInfos.SubscribeBlocking) THEN
	IF NOT BuildSubscribePaket(PaketData:= OutData[SendInfos.SubscribeIndex].InDataFromFb) THEN
		SendInfos.SubscribeBlocking := TRUE;
	ELSE
		SendInfos.SubscribeBlocking := FALSE;
		SendInfos.SubscribeNeeded := FALSE;
		OutData[SendInfos.SubscribeIndex].TimeOutStarted := TRUE;
		OutData[SendInfos.SubscribeIndex].step := STEPS_OUT.WAIT_SUBACK;
	END_IF
END_IF
//send pending Publish 
IF SendInfos.PublishBlocking THEN
	IF BuildPublishPaket(PaketData:= OutData[SendInfos.PublishBlockingIndex].InDataFromFb) THEN
		SendInfos.PublishBlocking := FALSE;
		PublishSendDone(slot:=ADR(OutData[SendInfos.PublishBlockingIndex]));
	END_IF
END_IF

IF (PublishSendListCount > 0 AND NOT SomethingIsBlocking) THEN
	//handle pendig publisah packet
	//handle new publish packet
	FOR i := 0 TO PublishSendListCount - 1 DO
		IF NOT BuildPublishPaket(PaketData:= OutData[PublishSendList[i]].InDataFromFb) THEN
			SendInfos.PublishBlocking := TRUE;
			SendInfos.PublishBlockingIndex := PublishSendList[i];
			EXIT;
		ELSE 
			SendInfos.PublishBlocking := FALSE;
			PublishSendDone(slot:=ADR(OutData[PublishSendList[i]]));
		END_IF
	END_FOR
END_IF
                
END_METHOD

METHOD SendInData
  VAR_INPUT
    MQTT_IN_OUT : POINTER TO MQTT_IN_OUT;
  END_VAR
  VAR
    i : UINT;
  END_VAR
                  IF NOT SendFree THEN RETURN; END_IF

GVL_MQTT.ProgNum := PROG_NUM.SendInData;

IF NOT COM.S_BUF.SIZE = 0 THEN 
	CountInSendNotFree := CountInSendNotFree + 1;
END_IF

IF PubackSendListCount > 0 THEN
	//SendInfos.PubackNeeded := FALSE;
	FOR i := 0 TO PubackSendListCount - 1 DO
		IF NOT (COM.S_BUF.SIZE + SIZE_PUBACK > TRANSMIT_BUFFER_SIZE)  THEN
			COM.S_BUF.BUFFER[COM.S_BUF.SIZE] := MESSAGETYPE.PUBACK;
			COM.S_BUF.BUFFER[COM.S_BUF.SIZE + 1] := 2;//length of 2
			COM.S_BUF.BUFFER[COM.S_BUF.SIZE + 2] := OSCAT_BASIC.BYTE_OF_DWORD(in:= InData[PubackSendList[i]].PaketID, N:= 1);
			COM.S_BUF.BUFFER[COM.S_BUF.SIZE + 3] := OSCAT_BASIC.BYTE_OF_DWORD(in:= InData[PubackSendList[i]].PaketID, N:= 0);
			COM.S_BUF.SIZE := COM.S_BUF.SIZE + SIZE_PUBACK;//Paket size allways 4!
			InData[PubackSendList[i]].step := STEPS_IN.WAIT_DATA;
			MqttsDoneIo := MqttsDoneIo + 1;	
		ELSE
			EXIT;
		END_IF
	END_FOR
	
END_IF

IF PubcompSendListCount > 0 THEN
	//SendInfos.PubcompNeeded := FALSE;
	FOR i := 0 TO PubcompSendListCount - 1 DO
		IF NOT (COM.S_BUF.SIZE + SIZE_PUBCOMP > TRANSMIT_BUFFER_SIZE) THEN	
			COM.S_BUF.BUFFER[COM.S_BUF.SIZE] := MESSAGETYPE.PUBCOMP;
			COM.S_BUF.BUFFER[COM.S_BUF.SIZE + 1] := 2;//length of 2
			COM.S_BUF.BUFFER[COM.S_BUF.SIZE + 2] := OSCAT_BASIC.BYTE_OF_DWORD(in:= InData[PubcompSendList[i]].PaketID, N:= 1);
			COM.S_BUF.BUFFER[COM.S_BUF.SIZE + 3] := OSCAT_BASIC.BYTE_OF_DWORD(in:= InData[PubcompSendList[i]].PaketID, N:= 0);
			COM.S_BUF.SIZE := COM.S_BUF.SIZE + SIZE_PUBCOMP;//Paket size allways 4!
			InData[PubcompSendList[i]].step := STEPS_IN.WAIT_DATA;
			MqttsDoneIo := MqttsDoneIo + 1;
		ELSE
			EXIT;
		END_IF
	END_FOR
END_IF

IF PubrecSendListCount > 0 THEN
	FOR i := 0 TO PubrecSendListCount - 1 DO
		IF NOT (COM.S_BUF.SIZE + SIZE_PUBREC > TRANSMIT_BUFFER_SIZE) THEN
			//SendInfos.PubrecNeeded := FALSE;
			COM.S_BUF.BUFFER[COM.S_BUF.SIZE] := MESSAGETYPE.PUBREC;
			COM.S_BUF.BUFFER[COM.S_BUF.SIZE + 1] := 2;//length of 2
			COM.S_BUF.BUFFER[COM.S_BUF.SIZE + 2] := OSCAT_BASIC.BYTE_OF_DWORD(in:= InData[PubrecSendList[i]].PaketID, N:= 1);
			COM.S_BUF.BUFFER[COM.S_BUF.SIZE + 3] := OSCAT_BASIC.BYTE_OF_DWORD(in:= InData[PubrecSendList[i]].PaketID, N:= 0);
			COM.S_BUF.SIZE := COM.S_BUF.SIZE + SIZE_PUBREC;//Paket size allways 4!
			InData[PubrecSendList[i]].step := STEPS_IN.WAIT_PUBREL;
			InData[PubrecSendList[i]].TimeOutStarted := TRUE;
		ELSE
			EXIT;
		END_IF
	END_FOR
END_IF

                
END_METHOD

METHOD ParseIncoming
  VAR_INPUT
    MQTT_IN_OUT : POINTER TO MQTT_IN_OUT;
  END_VAR
  VAR
    I : UINT;
    j : UINT;
    idx : UINT := 0;
    RecivePakteType : MESSAGETYPE;  (* idxFromParsePublish:UINT := 0; *)
    RecivePaketID : WORD;
    BufferMoveDone : BOOL;
    PaketFound : BOOL;
  END_VAR
                  GVL_MQTT.ProgNum := PROG_NUM.ParseIncomming;
IF COM.R_BUF.SIZE > 0 THEN
	REPEAT
		
		PaketFound := FALSE;
		HelperLastPaktetForUnkownPaket := RecivePakteType;
		RecivePakteType := COM.R_BUF.BUFFER[idx] AND 16#F0;
		 
		CASE RecivePakteType OF
			MESSAGETYPE.PUBLISH:
			//new way, move every publish to recive buffer, and then pars it.
			//outgoing payload pointer is then set to start of payload in the buffer....
				//don't use check buffer here, make all in Parse Publish....
				BufferMoveDone := CheckLenghtBuffer(IdxIn:= idx);
				IF NOT BufferMoveDone THEN
					
					idx := ParseIncomingPublish(MQTT_IN_OUT:= MQTT_IN_OUT, idx:= idx,
											BufferIn:= ADR(COM.R_BUF.BUFFER), BufferSize:= COM.R_BUF.SIZE,
											NetworkBuffer:= TRUE);

				END_IF
			MESSAGETYPE.PUBREL:
				BufferMoveDone := CheckLenghtBuffer(IdxIn:= idx);
				IF NOT BufferMoveDone THEN
					//get Paket ID
					RecivePaketID := DWORD_TO_WORD(OSCAT_BASIC.DWORD_OF_BYTE(B3:= 0, B2:= 0, 
						B1:= COM.R_BUF.BUFFER[idx + 2],
						B0:= COM.R_BUF.BUFFER[idx + 3]));
					//find Paket
					FOR i := 0 TO MyConstants.QoS_BUFFER_SIZE - 1 DO
						IF InData[i].PaketID = RecivePaketID THEN
							InData[i].step := STEPS_IN.SEND_PUBCOMP;
							InData[i].TimeOutStarted := FALSE;
							PubcompOrderIndexCounter := PubcompOrderIndexCounter;
							InData[i].PUBCOMPOrder := PubcompOrderIndexCounter;
							PaketFound := TRUE;
							EXIT;
						END_IF
						//
					END_FOR
					IF NOT PaketFound THEN
						CountRecivePubrelUnknown := CountRecivePubrelUnknown + 1;
					END_IF
					idx := idx + SIZE_PUBREL;
				END_IF
			MESSAGETYPE.PINGRESP:
				ResetPingTime();
				PingRequestet := FALSE;
				OutData[PingSlot].step := STEPS_OUT.WAIT_DATA;//can get new data
				OutData[PingSlot].TimeOutStarted := FALSE;
				idx := idx + SIZE_PINGRESP;
			MESSAGETYPE.UNSUBACK:
				BufferMoveDone := CheckLenghtBuffer(IdxIn:= idx);
				IF NOT BufferMoveDone THEN
					//get Paket ID
					RecivePaketID := DWORD_TO_WORD(OSCAT_BASIC.DWORD_OF_BYTE(B3:= 0, B2:= 0, 
						B1:= COM.R_BUF.BUFFER[idx + 2],
						B0:= COM.R_BUF.BUFFER[idx + 3]));
					//find Paket
					FOR i := 0 TO MyConstants.QoS_BUFFER_SIZE - 1 DO
						IF OutData[i].step = STEPS_OUT.WAIT_UNSUBACK THEN //make sure pointer is vailid
							IF OutData[i].InDataFromFb^.PaketId = RecivePaketID THEN
								OutData[i].InDataFromFb^.SendSucsess := TRUE;
								OutData[i].step := STEPS_OUT.WAIT_DATA;//can get new data
								OutData[i].TimeOutStarted := FALSE;
								MqttsDoneIo := MqttsDoneIo + 1;
								PaketFound := TRUE;
								//now kick of Callback
								FOR j := 0 TO CALLBACKS_BUFFER_SIZE - 1 DO
									IF SubscribeCallbacks[j].FbId = OutData[i].InDataFromFb^.FbId THEN
										//callback found, now kill it...
										SubscribeCallbacks[j].free := TRUE;
										SubscribeCallbacks[j].FbId := 0;
										EXIT;
									END_IF
								END_FOR
								EXIT;
							END_IF
						END_IF
						//
					END_FOR
					IF NOT PaketFound THEN
						CountReciveUnsubackUnknown := CountReciveUnsubackUnknown + 1;
					END_IF
					idx := idx + SIZE_UNSUBACK;	
				END_IF
				
			MESSAGETYPE.SUBACK:
				BufferMoveDone := CheckLenghtBuffer(IdxIn:= idx);
				IF NOT BufferMoveDone THEN
					//get Paket ID
					RecivePaketID := DWORD_TO_WORD(OSCAT_BASIC.DWORD_OF_BYTE(B3:= 0, B2:= 0, 
						B1:= COM.R_BUF.BUFFER[idx + 2],
						B0:= COM.R_BUF.BUFFER[idx + 3]));
					//find Paket
					FOR i := 0 TO MyConstants.QoS_BUFFER_SIZE - 1 DO
						IF OutData[i].step = STEPS_OUT.WAIT_SUBACK THEN //make sure pointer is vailid
							IF OutData[i].InDataFromFb^.PaketId = RecivePaketID THEN
								OutData[i].InDataFromFb^.SendSucsess := TRUE;
								OutData[i].InDataFromFb^.SubackQoS := COM.R_BUF.BUFFER[idx + 4];
								OutData[i].step := STEPS_OUT.WAIT_DATA;//can get new data
								OutData[i].TimeOutStarted := FALSE;
								MqttsDoneIo := MqttsDoneIo + 1;
								PaketFound := TRUE;
								//now register callback:
								FOR j := 0 TO CALLBACKS_BUFFER_SIZE - 1 DO
									IF SubscribeCallbacks[j].free THEN
										SubscribeCallbacks[j].free := FALSE;
										SubscribeCallbacks[j].Callback := OutData[i].InDataFromFb^.Callback;
 										SubscribeCallbacks[j].FbId := OutData[i].InDataFromFb^.FbId;
										SubscribeCallbacks[j].SplitTopic := OutData[i].InDataFromFb^.SplitTopic;
										SubscribeCallbacks[j].ExpectingString := OutData[i].InDataFromFb^.ExpectingString;
										EXIT;
									END_IF
								END_FOR
								IF j = CALLBACKS_BUFFER_SIZE THEN
									//no callback slot free
									OutData[i].InDataFromFb^.CallbackError := TRUE;
								END_IF
								EXIT;
							END_IF
						END_IF
						//
					END_FOR
					IF NOT PaketFound THEN
						CountReciveSubackUnknown := CountReciveSubackUnknown + 1;
					END_IF
					idx := idx + SIZE_SUBACK;//only one QoS response expected
				END_IF
			MESSAGETYPE.PUBACK:
				BufferMoveDone := CheckLenghtBuffer(IdxIn:= idx);
				IF NOT BufferMoveDone THEN
					//get Paket ID
					RecivePaketID := DWORD_TO_WORD(OSCAT_BASIC.DWORD_OF_BYTE(B3:= 0, B2:= 0, 
						B1:= COM.R_BUF.BUFFER[idx + 2],
						B0:= COM.R_BUF.BUFFER[idx + 3]));
					//find Paket
					FOR i := 0 TO MyConstants.QoS_BUFFER_SIZE - 1 DO
						IF OutData[i].step = STEPS_OUT.WAIT_PUBACK THEN //make sure pointer is vailid
							IF OutData[i].InDataFromFb^.PaketId = RecivePaketID THEN
								OutData[i].InDataFromFb^.SendSucsess := TRUE;
								OutData[i].step := STEPS_OUT.WAIT_DATA;//can get new data
								OutData[i].TimeOutStarted := FALSE;
								MqttsDoneIo := MqttsDoneIo + 1;
								Publishsunacknowledged := Publishsunacknowledged - 1;
								PaketFound := TRUE; 
								EXIT;
							END_IF
						END_IF
						//
					END_FOR
					IF NOT PaketFound THEN
						CountRecivePubackUnknown := CountRecivePubackUnknown + 1;
					END_IF
					idx := idx + SIZE_PUBACK;
				END_IF
			MESSAGETYPE.PUBREC:
				BufferMoveDone := CheckLenghtBuffer(IdxIn:= idx);
				IF NOT BufferMoveDone THEN
					//get Paket ID
					RecivePaketID := DWORD_TO_WORD(OSCAT_BASIC.DWORD_OF_BYTE(B3:= 0, B2:= 0, 
						B1:= COM.R_BUF.BUFFER[idx + 2],
						B0:= COM.R_BUF.BUFFER[idx + 3]));
					//find Paket
					FOR i := 0 TO MyConstants.QoS_BUFFER_SIZE - 1 DO
						IF OutData[i].step = STEPS_OUT.WAIT_PUBREC THEN //make sure pointer is vailid
							IF OutData[i].InDataFromFb^.PaketId = RecivePaketID THEN
								IF NOT OutData[i].InDataFromFb^.DUP THEN
									//increase only at first handle 
									PubrelOrderIndexCounter := PubrelOrderIndexCounter + 1;
									OutData[i].PUBRECOrder := PubrelOrderIndexCounter;
								END_IF
								OutData[i].step := STEPS_OUT.SEND_PUBREL;
								OutData[i].TimeOutStarted := FALSE;
								PaketFound := TRUE; 
								EXIT;
							END_IF
						END_IF
						//
					END_FOR
					IF NOT PaketFound THEN
						CountRecivePubrecUnknown := CountRecivePubrecUnknown + 1;
					END_IF
					idx := idx + SIZE_PUBREC;
				END_IF
			MESSAGETYPE.PUBCOMP:
				BufferMoveDone := CheckLenghtBuffer(IdxIn:= idx);
				IF NOT BufferMoveDone THEN
					//get Paket ID
					RecivePaketID := DWORD_TO_WORD(OSCAT_BASIC.DWORD_OF_BYTE(B3:= 0, B2:= 0, 
						B1:= COM.R_BUF.BUFFER[idx + 2],
						B0:= COM.R_BUF.BUFFER[idx + 3]));
					//find Paket
					FOR i := 0 TO MyConstants.QoS_BUFFER_SIZE - 1 DO
						IF OutData[i].step = STEPS_OUT.WAIT_PUBCOMP THEN //make sure pointer is vailid
							IF OutData[i].InDataFromFb^.PaketId = RecivePaketID THEN
								OutData[i].InDataFromFb^.SendSucsess := TRUE;
								OutData[i].step := STEPS_OUT.WAIT_DATA;//can get new data
								OutData[i].TimeOutStarted := FALSE;
								MqttsDoneIo := MqttsDoneIo + 1;
								Publishsunacknowledged := Publishsunacknowledged - 1;
								PaketFound := TRUE;
								EXIT;
							END_IF
						END_IF
						//
					END_FOR
					IF NOT PaketFound THEN
						CountRecivePubcompUnknown := CountRecivePubcompUnknown + 1;
					END_IF
					idx := idx + SIZE_PUBCOMP;			
				END_IF
			ELSE
				//unknown paket, reset buffer....
				//standard wants to disconnect....
				{info 'unkown packet, disconnect'}
				LastPaktetForUnkownPaket := HelperLastPaktetForUnkownPaket;
				COM.R_BUF.SIZE := 0;	
				//unknown paket recived
				NotKnownPaket := COM.R_BUF.BUFFER[0] AND 16#F0;
				//alway reset recive!
				COM.MQTT_RCV_STATE := BYTE#0;//recive zurücksetzten
				COM.R_BUF.SIZE := 0;
				CountUnkownPaket := CountUnkownPaket + 1;	
		END_CASE
	UNTIL
		idx >= COM.R_BUF.SIZE OR BufferMoveDone
	END_REPEAT
	IF NOT BufferMoveDone THEN
		COM.R_BUF.SIZE := 0;
		COM.MQTT_RCV_STATE := BYTE#0;//recive zurücksetzten	
	END_IF
	
END_IF
                
END_METHOD

METHOD ParseIncomingPublish : UINT
  VAR_INPUT
    MQTT_IN_OUT : POINTER TO MQTT_IN_OUT;
    idx : UINT;  (* pos of paket in buffer *)
    BufferIn : POINTER TO BYTE;  (* give here the buffer were the full packet is... *)
    NetworkBuffer : BOOL;  (* works on network buffer --> need memmove in Output *)
    BufferSize : UDINT;  (* size of buffer, bytes occupied *)
  END_VAR
  VAR
    i : UINT;
    PaketFound : BOOL;
    PaketIndex : UINT;
    FreeSlot : UINT;
    FreeSlotFound : BOOL;
    RecivePaketID : WORD;
    ReciveQoSLevel : QoS;
    TopicSize : UINT;
    OutData : BOOL;  (* Output the Data, Tru if Data can be outputted *)
    RemainingLength : REMAINING_LENGTH_RETURN;
    PayloadPosStart : UDINT;
    TopicPosStart : UDINT;
    PayloadSize : UDINT;
    FollowingDataBuffer : ARRAY[0..1] OF BYTE;  (* NextPosReciveBuffer : UINT; *)
    PayloadMoved : BOOL;
  END_VAR
                  ParseIncomingPublish := 0;//if return is zero, buffer move has been done,
CounterPublishRecivedForMonitor := CounterPublishRecivedForMonitor + 1;
GVL_MQTT.ProgNum := PROG_NUM.ParsePublish;
//get remaining length
RemainingLength := GetRemainingLength(BufferIn, pos := idx,BuffSize := BufferSize);
TopicPosStart := RemainingLength.IndexAfterRemainingLength + 2;
ReciveQoSLevel := SHR(BufferIn[idx] AND 2#110,1);

TopicSize := DWORD_TO_WORD(OSCAT_BASIC.DWORD_OF_BYTE(B3:= 0, B2:= 0,
						 B1:= BufferIn[RemainingLength.IndexAfterRemainingLength],
						 B0:= BufferIn[RemainingLength.IndexAfterRemainingLength+1]));
IF RemainingLength.Error THEN
	//throw away paket on length error
	COM.MQTT_RCV_STATE := BYTE#0;//recive zurücksetzten
	//need to set size to zero, so no further parsing...
	COM.R_BUF.SIZE := 0;
	CountLengthErrors := CountLengthErrors;
	//on standard i MUST diconnect!!!
	DoDisconnect := TRUE;
	
	RETURN;
END_IF
//publish recived, size is handleable
IF ReciveQoSLevel = QoS.AtMostOnce THEN
	//Nothing to do, just out the Payload and Topic
	OutData := TRUE;
	PayloadSize := RemainingLength.RemainingLength - TopicSize - 2;//2 for Size Encoding
	PayloadPosStart := RemainingLength.IndexAfterRemainingLength + TopicSize + 2;//2 for Size Encoding
ELSE
	//get Paket ID
	RecivePaketID := DWORD_TO_WORD(OSCAT_BASIC.DWORD_OF_BYTE(B3:= 0, B2:= 0, 
		B1:= BufferIn[RemainingLength.IndexAfterRemainingLength + TopicSize + 2],//+ 2 for Topic Length
		B0:= BufferIn[RemainingLength.IndexAfterRemainingLength + TopicSize + 3]));
	//2 for size of Paket identifier
	PayloadSize := RemainingLength.RemainingLength - TopicSize - 4;//2 for size of topic  and 2 for message id
	PayloadPosStart := RemainingLength.IndexAfterRemainingLength + TopicSize + 4;//2 for size of topic and 2 for message id
	
	//QoS stuff
	FOR i := 0 TO MyConstants.QoS_BUFFER_SIZE - 1 DO
		IF InData[i].PaketID = RecivePaketID AND InData[i].step <> STEPS_IN.WAIT_DATA THEN
			PaketIndex := i;
			PaketFound := TRUE;
			
		END_IF
		IF InData[i].step = STEPS_IN.WAIT_DATA AND NOT FreeSlotFound THEN
			FreeSlot := i;
			FreeSlotFound := TRUE;
		END_IF
		IF FreeSlotFound AND PaketFound THEN
			EXIT;//exit if slot and paket found
		END_IF
	END_FOR
	IF NOT PaketFound THEN
		IF FreeSlotFound THEN
			//Paket ist not to be awnserd --> first occurence
			InData[FreeSlot].CountPubrecRepeat := 0;
			InData[FreeSlot].QoS := ReciveQoSLevel;
			InData[FreeSlot].PaketID := RecivePaketID;
			IncomingPublishOrderIndexCounter := IncomingPublishOrderIndexCounter + 1;
			InData[FreeSlot].PUBLISHOrder := IncomingPublishOrderIndexCounter;
			OutData := TRUE;
			CountRecivedPublishs := CountRecivedPublishs + 1;
		ELSE
			//no more slots free
			{info 'no more slots free, what shall we do???'}
			//at all this is fine....
			DoDisconnect := TRUE;
			
		END_IF
	ELSE
		CountRepeatPublishRecive := CountRepeatPublishRecive + 1;
	END_IF
	CASE InData[FreeSlot].QoS OF
		QoS.AtLeastOnce:
			InData[FreeSlot].step := STEPS_IN.SEND_PUBACK;
		QoS.ExactlyOnce:
			InData[FreeSlot].step := STEPS_IN.SEND_PUBREC;
	END_CASE
END_IF

IF RemainingLength.RemainingLength > (COM_CONFIG.MaxTopicElementSize * COM_CONFIG.MaxTopicLevels + COM_CONFIG.MaxPayloadSize) OR 
	TopicSize > (COM_CONFIG.MaxTopicElementSize * COM_CONFIG.MaxTopicLevels) OR
	PayloadSize > COM_CONFIG.MaxPayloadSize THEN
	{info 'check here if to disconnect'}
	//paket to big for my Strings, but do QoS stuff!!!! no standard, standard wants disconnect!
	CountToBigTopics := CountToBigTopics  + 1;
	{info 'check if last to big topic is to saved, or just take memmove'}
	(*LastToBigTopic := OSCAT_BASIC.BUFFER_TO_STRING(PT:= ADR(BufferIn[idx]), SIZE:= BufferSize,
						START:= RemainingLength.IndexAfterRemainingLength + 2,
						STOP:= RemainingLength.IndexAfterRemainingLength + TopicSize);*)
	OutData := FALSE;//reset out Data....
END_IF


//now set idx to next packet
ParseIncomingPublish := UDINT_TO_UINT(PayloadPosStart + PayloadSize);

IF OutData THEN
		
		//new approch: in buffer for big packets we can move as we want. in network buffer, we can move topic
		//without trobble down, length information isn't needed anymore. if we move in network buffer we store 
		//the following two bytes of payload, making the output and there after we restore them.
		//this we do in buffer for big packets too, because it isn't expensive
		//but we have to be aware if the payload is near the buffer end, then we have to move it down...

		//we need to check if  
		
		//IF NOT NetworkBuffer THEN //in network buffer, we have to set an termination
		PayloadMoved := FALSE;	
		//first check if payload needs to be moved, because it is at the buffer end
		IF NetworkBuffer THEN
			IF ReciveQoSLevel = QoS.AtMostOnce THEN//if QoS zero, we need to move, because space for packet ID is missing...
				//check which is smaller, this is to be moved....
				IF TopicSize < PayloadSize THEN
					//move Topic down
					MEM.MemMove(pSource:= ADR(BufferIn[TopicPosStart]), pDestination:= ADR(BufferIn[TopicPosStart - 1]), uiNumberOfBytes:= TopicSize);
					TopicPosStart := TopicPosStart - 1;//now topic resits one deeper
				ELSE
					IF idx + PayloadPosStart + PayloadSize > MyConstants.NETWORK_BUFFER_LONG_SIZE THEN
						//need to move payload and topic, I'm at the top border of network buffer
						//should be very rare....
						//SysMem23.SysMemMove30(pDest:= ADR(BufferIn[TopicPosStart - 2]), pSrc:= ADR(BufferIn[TopicPosStart]), diCount:= TO_DINT(TopicSize));
						SysMem.SysMemMove(pDest:= ADR(BufferIn[TopicPosStart - 2]), pSrc:= ADR(BufferIn[TopicPosStart]), udiCount:= TO_UDINT(TopicSize));
						//SysMem23.SysMemMove30(pDest:= ADR(BufferIn[PayloadPosStart - 1]), pSrc:= ADR(BufferIn[PayloadPosStart]), diCount:= TO_DINT(PayloadSize));
						SysMem.SysMemMove(pDest:= ADR(BufferIn[PayloadPosStart - 1]), pSrc:= ADR(BufferIn[PayloadPosStart]), udiCount:= TO_UDINT(PayloadSize));
						//change Topic Pointer...
						TopicPosStart := TopicPosStart - 2;
						//change Payload Pointer
						PayloadPosStart := PayloadPosStart - 1;
					ELSE
						//first, save following data
						//move Payload up
						PayloadMoved := TRUE;
						FollowingDataBuffer[0] := BufferIn[PayloadPosStart + PayloadSize];
						SysMem.SysMemMove(pDest:= ADR(BufferIn[PayloadPosStart + 1]), pSrc:= ADR(BufferIn[PayloadPosStart]), udiCount:= TO_UDINT(PayloadSize));
						PayloadPosStart := PayloadPosStart + 1;//payload now resits one higher
					END_IF
				END_IF
			END_IF
			
			//alway set termination for payload because it could be a string
			FollowingDataBuffer[1] := BufferIn[PayloadPosStart + PayloadSize]; 
			BufferIn[PayloadPosStart + PayloadSize] := 0;	
			//now set termination, if not QoS zero, overwrite PacketID
			BufferIn[TopicPosStart + TopicSize] := 0;
			//END_IF
			OutputPublish(
				PayloadSize:= PayloadSize, 
				PayloadPos:= ADR(BufferIn[PayloadPosStart]), 
				TopicSize:= TopicSize, 
				TopicPos:= ADR(BufferIn[TopicPosStart]), 
				MQTT_IN_OUT:= MQTT_IN_OUT);
			//restore data after payload
			BufferIn[PayloadPosStart + PayloadSize] := FollowingDataBuffer[1];
			//END_IF

		ELSE
			
		//here we are not in the network buffer, borders don't care and following bytes doesn't matter.
			IF ReciveQoSLevel = QoS.AtMostOnce THEN//if QoS zero, we need to move, because space for packet ID is missing...
				//check which is smaller, this is to be moved....
				IF TopicSize < PayloadSize THEN
					//move Topic down
					MEM.MemMove(pSource:= ADR(BufferIn[TopicPosStart]), pDestination:= ADR(BufferIn[TopicPosStart - 1]), uiNumberOfBytes:= TopicSize);
					TopicPosStart := TopicPosStart - 1;//now topic resits one deeper
				ELSE
					//move Payload up
					SysMem.SysMemMove(pDest:= ADR(BufferIn[PayloadPosStart + 1]), pSrc:= ADR(BufferIn[PayloadPosStart]), udiCount:= TO_UDINT(PayloadSize));
					PayloadPosStart := PayloadPosStart + 1;//payload now resits one higher
				END_IF
			END_IF
			//alway set termination for payload because it could be a string
			BufferIn[PayloadPosStart + PayloadSize] := 0;	
			//now set termination, if not QoS zero, overwrite PacketID
			BufferIn[TopicPosStart + TopicSize] := 0;
			//END_IF
			OutputPublish(
				PayloadSize:= PayloadSize, 
				PayloadPos:= ADR(BufferIn[PayloadPosStart]), 
				TopicSize:= TopicSize, 
				TopicPos:= ADR(BufferIn[TopicPosStart]), 
				MQTT_IN_OUT:= MQTT_IN_OUT);
			
		END_IF
END_IF

IF PayloadMoved THEN 
	//if payload was moved, then content have to be rebuild
	BufferIn[PayloadPosStart + PayloadSize - 1] := FollowingDataBuffer[0];
END_IF
                
END_METHOD

METHOD CheckLenghtBuffer : BOOL
  VAR_INPUT
    IdxIn : UINT;
  END_VAR
  VAR
    RecivePakteType : MESSAGETYPE;
    RemainingLength : REMAINING_LENGTH_RETURN;
    NeedBufferMove : BOOL;
  END_VAR
                  CheckLenghtBuffer := FALSE;

RecivePakteType := COM.R_BUF.BUFFER[IdxIn] AND 16#F0;

NeedBufferMove := FALSE;

CASE RecivePakteType OF

	MESSAGETYPE.PUBLISH:
		IF IdxIn + 1 > COM.R_BUF.SIZE THEN//1 for max size of remaining length
			CheckLenghtBuffer := TRUE;//let this, if just one ore two bytes of publish packet was recived
		ELSE
			//size big enough to test remaining lengt, inside testing of bytes....
			RemainingLength := GetRemainingLength(ADR(COM.R_BUF.BUFFER), pos := IdxIn, BuffSize:= COM.R_BUF.SIZE);
			//if paket to small for buffer, disconnect, remaining length is smaller then whole packet size
			IF RemainingLength.RemainingLength - 8 > MaxPublishPacketSize THEN
				{info 'make this to a parameter to chose disconnect or discharge'}
				DoDisconnect := TRUE;
				CheckLenghtBuffer := TRUE;
			ELSE 
				
				IF (IdxIn + RemainingLength.RemainingLength >= COM.R_BUF.SIZE) THEN
				//
				//move splited publish packet to buffer
					//IF SplitPublishLock THEN
						//move publish packet in network recive buffer
					NeedBufferMove := TRUE;			
					(*ELSE
						//buffer is locked(packet is published to application) so move splited data in recive buffer for next cycle...
						SplitPublishLength := RemainingLength.RemainingLength + RemainingLength.SizeRemainingLength + 1;//one byte for fixed packed header
						SplitPublishBufferSize := COM.R_BUF.SIZE - IdxIn;;//new splited publish
						MEM.MemMove(pSource:= ADR(COM.R_BUF.BUFFER[IdxIn]), pDestination:= SplitPublishBuffer, uiNumberOfBytes:= UDINT_TO_UINT(SplitPublishBufferSize));
						//clear in Buffer
						COM.R_BUF.SIZE := 0;
						PublishSplited := TRUE;
						CheckLenghtBuffer := TRUE;
					END_IF*)
				END_IF 				
			END_IF
		END_IF
	MESSAGETYPE.PUBREL:
		IF IdxIn + SIZE_PUBREL > COM.R_BUF.SIZE THEN
			NeedBufferMove := TRUE;
		END_IF
	MESSAGETYPE.UNSUBACK:
		IF IdxIn + SIZE_UNSUBACK > COM.R_BUF.SIZE THEN
			NeedBufferMove := TRUE;
		END_IF
	MESSAGETYPE.SUBACK:
		IF IdxIn + SIZE_SUBACK > COM.R_BUF.SIZE THEN
			NeedBufferMove := TRUE;
		END_IF
	MESSAGETYPE.PUBACK:
		IF IdxIn + SIZE_PUBACK > COM.R_BUF.SIZE THEN
			NeedBufferMove := TRUE;
		END_IF
	MESSAGETYPE.PUBREC:
		IF IdxIn + SIZE_PUBREC > COM.R_BUF.SIZE THEN
			NeedBufferMove := TRUE;
		END_IF
	MESSAGETYPE.PUBCOMP:
		IF IdxIn + SIZE_PUBCOMP > COM.R_BUF.SIZE THEN
			NeedBufferMove := TRUE;
		END_IF

END_CASE

IF NeedBufferMove THEN
	MoveBufferForSplitPaket(idx:= IdxIn);
	InBufferMoved := 1;
	CheckLenghtBuffer := TRUE;
ELSE
	InBufferMoved := 0;
	CountWaitForRestOfPaket := 0;
END_IF

IF InBufferMoved = 1 THEN
	CountWaitForRestOfPaket := CountWaitForRestOfPaket + 1;
END_IF

IF CountWaitForRestOfPaket > 1000 THEN
	//waited long for rest of paket, so reset...	
	//unknown paket, reset buffer....
	//standard wants to disconnect....
	{info 'TODO:check to make disconnect as parameter'}
	DoDisconnect := TRUE;
	COM.R_BUF.SIZE := 0;	
	//unknown paket recived
	NotKnownPaket := COM.R_BUF.BUFFER[0] AND 16#F0;
	//allway reset recive!
	COM.MQTT_RCV_STATE := BYTE#0;//recive zurücksetzten
	COM.R_BUF.SIZE := 0;
	CountWaitForRestOfPaket := 0;
	CountResetBufferIn := CountResetBufferIn + 1;
END_IF
                
END_METHOD

METHOD FB_Exit : BOOL
  VAR_INPUT
    bInCopyCode : BOOL;  (* TRUE: the exit method is called in order to leave the instance which will be copied afterwards (online change). *)
  END_VAR
                  destroy();

                
END_METHOD

METHOD destroy : BOOL
  VAR
    iu : UINT;
  END_VAR
                  //cannot decrease memmory usage here at reset, this will trigger an accsess violation on windows... so usag maybe coruptetd! 
//DynMemUsagePointer^ := DynMemUsagePointer^ - (MaxPublishPacketSize + SPLIT_PUBLISH_BUFFER_ADDITIONAL_RAM);
MySplitTopic.destroy();
GVL_MQTT.ProgNum := PROG_NUM.DESTROY_HANDLE_MQTT;
{info 'semaphore'}

{warning disable C0033}
//SysMem23.SysMemFree(dwAddress:= SplitPublishBuffer, dwSize:= MaxPublishPacketSize + SPLIT_PUBLISH_BUFFER_ADDITIONAL_RAM);
__DELETE(SplitPublishBuffer);
{warning restore C0033}

                
END_METHOD

